// TIA Portal project "Braccio robotico_man_aut_completo_02_5AROB" (V16)

(* hardware
DEVICE "S7-1200 station_1"  S7-1200 Station
   slot 0: "Telaio di montaggio_0"  S7-1200 Rack  Rack  V1.0
   slot 1: "PLC_1"  CPU 1215C AC/DC/Rly  6ES7 215-1BG40-0XB0  V4.2
DEVICE "HMI_1"  KTP700 Basic PN
   slot 0: "HMI_1"  KTP700 Basic PN  6AV2 123-2GB03-0AX0  16.0.0.0
   slot 1: "HMI_RT_1"  KTP700 Basic PN  6AV2 123-2GB03-0AX0  16.0.0.0
   slot 5: "HMI_1.IE_CP_1"  PROFINET Interface  16.0.0.0
      slot 1: "Interfaccia_1 PROFINET"  PROFINET Interface
         slot 1: "Porta_1"  Port
*)

// ===== PLC "PLC_1"  CPU 1215C AC/DC/Rly =====

VAR_GLOBAL   // PLC tag table "Tabella variabili asse vericale"
   "SQ_alto_riferimento per lo zero" AT %I0.3 : Bool;
   "Impulsi contati dall'encoder verticale" AT %ID1000 : DWord;
   "Salita manuale" AT %M0.0 : Bool;
   "Discesa manuale" AT %M0.1 : Bool;
   "attivazione back to home" AT %M0.2 : Bool;
   "attivazione posizionamento automatico_vert" AT %M1.0 : Bool;
   "posizionamento automatico raggiunto_vert" AT %M1.1 : Bool;
   "posizionamento fuori tolleranza_vert" AT %M1.2 : Bool;
   "salita automatica" AT %M1.3 : Bool;
   "discesa automatica" AT %M1.4 : Bool;
   "Salita asse Z" AT %Q0.7 : Bool;
   "Discesa asse Z" AT %Q0.6 : Bool;
   "appoggio clock" AT %M1.6 : Bool;
   "Passo 4" AT %M30.5 : Bool;
   "Passo 5" AT %M30.6 : Bool;
   "Passo 6" AT %M30.7 : Bool;
   "Passo 7" AT %M31.0 : Bool;
   "Passo 8" AT %M31.1 : Bool;
   "Passo 9" AT %M31.2 : Bool;
   "Passo 10" AT %M31.3 : Bool;
END_VAR

VAR_GLOBAL   // PLC tag table "Tabella variabili rotazione"
   "SQ_rot_oraria_riferimento per lo zero" AT %I0.7 : Bool;
   "Impulsi contati dall'encoder rotazione" AT %ID1004 : DWord;
   "rotazione oraria manuale" AT %M2.0 : Bool;
   "rotazione antioraria manuale" AT %M2.1 : Bool;
   "attivazione back to home rotazione" AT %M2.2 : Bool;
   "attivazione posizionamento automatico_rot" AT %M3.0 : Bool;
   "posizionamento automatico raggiunto_rot" AT %M3.1 : Bool;
   "posizionamento fuori tolleranza_rot" AT %M3.2 : Bool;
   "rotazione oraria automatica" AT %M3.3 : Bool;
   "rotazione antioraria automatica" AT %M3.4 : Bool;
   "Rotazione oraria" AT %Q0.0 : Bool;
   "Rotazione antioraria" AT %Q0.1 : Bool;
END_VAR

VAR_GLOBAL   // PLC tag table "Tabella variabili braccio"
   "SQ_indietro_orizzontale" AT %I1.0 : Bool;
   "conteggio impulsi orizzontali" AT %MD5 : DInt;
   "avanti braccio manuale" AT %M4.0 : Bool;
   "indietro braccio manuale" AT %M4.1 : Bool;
   "attivazione back to home orizzontale" AT %M4.2 : Bool;
   "attivazione posizionamento automatico_orizzontale" AT %M4.3 : Bool;
   "posizionamento automatico raggiunto_orizzontale" AT %M4.4 : Bool;
   "posizionamento fuori tolleranza_orizzontale" AT %M4.5 : Bool;
   "avanti braccio in automatico" AT %M4.6 : Bool;
   "indietro braccio in automatico" AT %M4.7 : Bool;
   "Avanti braccio" AT %Q0.4 : Bool;
   "Indietro braccio" AT %Q0.5 : Bool;
   "SQ_impulsivo_orizzontale" AT %I1.1 : Bool;
END_VAR

VAR_GLOBAL   // PLC tag table "Tabella variabili pinza"
   "SQ_pinza_aperta" AT %I0.2 : Bool;
   "chiusura pinza manuale" AT %M10.0 : Bool;
   "apertura pinza manuale" AT %M10.1 : Bool;
   "attivazione back to home pinza" AT %M10.2 : Bool;
   "attivazione posizionamento automatico_pinza" AT %M10.3 : Bool;
   "posizionamento automatico raggiunto_pinza" AT %M10.4 : Bool;
   "posizionamento fuori tolleranza_pinza" AT %M10.5 : Bool;
   "chiusura pinza automatico" AT %M10.6 : Bool;
   "apertura pinza automatico" AT %M10.7 : Bool;
   "Chiusura pinza" AT %Q0.3 : Bool;
   "Apertura pinza" AT %Q0.2 : Bool;
   "conteggio impulsi pinza" AT %MD11 : DInt;
   "SQ_impulsivo_pinza" AT %I0.6 : Bool;
END_VAR

VAR_GLOBAL   // PLC tag table "Tabella variabili_ciclo_automatico"
   "condizioni_iniziali_ok" AT %M50.0 : Bool;
   "Passo 0" AT %M30.0 : Bool;
   "Passo 1" AT %M30.1 : Bool;
   "Passo 2" AT %M30.2 : Bool;
   "Passo 3" AT %M30.3 : Bool;
END_VAR

DATA_BLOCK "Blocco_dati_encoder_verticale"   // DB1
{ S7_Optimized_Access := 'TRUE' }
VERSION : 0.1
   VAR
      "posizione vericale in mm" : DInt;
      "setpoint verticale" : DInt;
      "tolleranza positiva verticale" : DInt;
      "tolleranza negativa verticale" : DInt;
      "appoggio ID1000" : DInt;
   END_VAR
BEGIN
END_DATA_BLOCK

DATA_BLOCK "Blocco_dati_HMI_verticale"   // DB2
{ S7_Optimized_Access := 'TRUE' }
VERSION : 0.1
   VAR
      jog_emergenza : Bool;
      jog_selettore_man_aut : Bool;
      jog_salita_braccio : Bool;
      jog_discesa_braccio : Bool;
      jog_back_to_home : Bool;
      setpoint_1 : DInt;
      setpoint_2 : DInt;
      setpoint_3 : DInt;
      setpoint_4 : DInt;
   END_VAR
BEGIN
END_DATA_BLOCK

DATA_BLOCK "Blocco_dati_HMI_automatico"   // DB3
{ S7_Optimized_Access := 'TRUE' }
VERSION : 0.1
   VAR
      jog_start_automatico : Bool;
      jog_ripristino : Bool;
   END_VAR
BEGIN
END_DATA_BLOCK

DATA_BLOCK "Blocco_dati_encoder_rotazione"   // DB6
{ S7_Optimized_Access := 'TRUE' }
VERSION : 0.1
   VAR
      "setpoint rotazione" : DInt;
      "tolleranza positiva rotazione" : DInt;
      "tolleranza negativa rotazione" : DInt;
      "posizione rotazione in gradi" : DInt;
      "appoggio ID1004" : DInt;
   END_VAR
BEGIN
END_DATA_BLOCK

DATA_BLOCK "Blocco_dati_HMI_rotazione"   // DB7
{ S7_Optimized_Access := 'TRUE' }
VERSION : 0.1
   VAR
      jog_rotazione_oraria : Bool;
      jog_rotazione_antioraia : Bool;
      jog_back_to_home_rotazione : Bool;
      jog_posizionamento_automatico_rot : Bool;
      setpoint_1 : DInt;
      setpoint_2 : DInt;
      setpoint_3 : DInt;
   END_VAR
BEGIN
END_DATA_BLOCK

DATA_BLOCK "Blocco_dati_contaimpulsi_braccio"   // DB8
{ S7_Optimized_Access := 'TRUE' }
VERSION : 0.1
   VAR
      "posizione orizzontale in mm" : DInt;
      "setpoint orizzontale" : DInt;
      "tolleranza positiva orizzontale" : DInt;
      "tolleranza negativa orizzontale" : DInt;
   END_VAR
BEGIN
END_DATA_BLOCK

DATA_BLOCK "Blocco_dati_contaimpulsi_pinza"   // DB9
{ S7_Optimized_Access := 'TRUE' }
VERSION : 0.1
   VAR
      "setpoint chiusura pinza" : DInt;
      "tolleranza positiva pinza" : DInt;
      "tolleranza negativa pinza" : DInt;
   END_VAR
BEGIN
END_DATA_BLOCK

DATA_BLOCK "Blocco_dati_HMI_braccio"   // DB10
{ S7_Optimized_Access := 'TRUE' }
VERSION : 0.1
   VAR
      jog_avanti_braccio : Bool;
      jog_indietro_braccio : Bool;
      jog_back_to_home_orizzontale : Bool;
      setpoint_1 : DInt;
      setpoint_2 : DInt;
      setpoint_3 : DInt;
   END_VAR
BEGIN
END_DATA_BLOCK

DATA_BLOCK "Blocco_dati_HMI_pinza"   // DB11
{ S7_Optimized_Access := 'TRUE' }
VERSION : 0.1
   VAR
      jog_chiusura_pinza : Bool;
      jog_apertura_pinza : Bool;
      jog_back_to_home_pinza : Bool;
      setpoint_1 : DInt;
      setpoint_2 : DInt;
   END_VAR
BEGIN
END_DATA_BLOCK

// folder: System blocks/Program resources

DATA_BLOCK "IEC_Counter_0_DB_1"   // DB12
{ S7_Optimized_Access := 'TRUE' }
AUTHOR : Simatic
FAMILY : IEC
NAME : CNTR
VERSION : 1.0
// stored: InstanceOfName IEC_COUNTER
"IEC_COUNTER"
BEGIN
END_DATA_BLOCK

DATA_BLOCK "TImer_passo9"   // DB13
{ S7_Optimized_Access := 'TRUE' }
AUTHOR : Simatic
FAMILY : IEC
NAME : IEC_TMR
VERSION : 1.0
// stored: InstanceOfName IEC_TIMER
"IEC_TIMER"
BEGIN
END_DATA_BLOCK

// folder: (top level)

FUNCTION "01_Calcoli_encoder_verticale" : Void   // FC1, LAD
{ S7_Optimized_Access := 'TRUE' }
VERSION : 0.1
BEGIN

REGION Network 1: Contatore veloce da configurare nelle proprietà della CPU
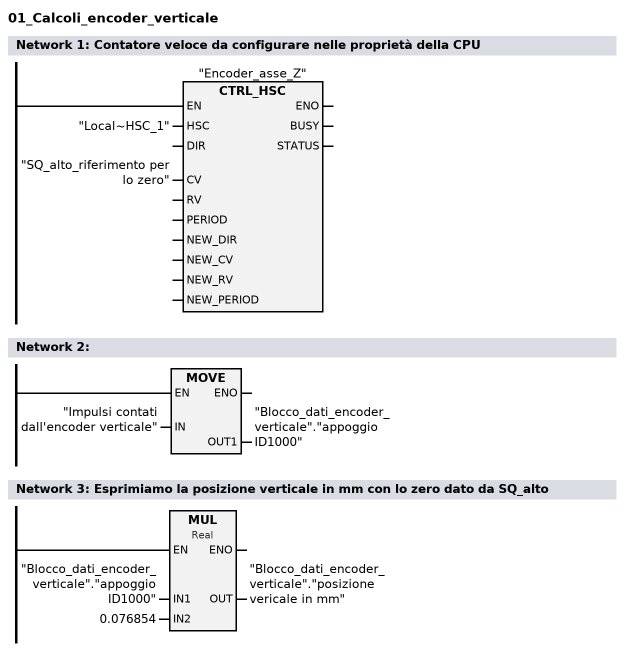
   "Encoder_asse_Z"(HSC := "Local~HSC_1", CV := "SQ_alto_riferimento per lo zero");   // CTRL_HSC
END_REGION

REGION Network 2
   RUNG wire#powerrail
      Move(in := "Impulsi contati dall'encoder verticale", out1 => "Blocco_dati_encoder_verticale"."appoggio ID1000")
   END_RUNG
   // the same network as SCL:
   "Blocco_dati_encoder_verticale"."appoggio ID1000" := "Impulsi contati dall'encoder verticale";
END_REGION

REGION Network 3: Esprimiamo la posizione verticale in mm con lo zero dato da SQ_alto
   RUNG wire#powerrail
      { S7_Templates := "SrcType := Real" } Mul(in1 := "Blocco_dati_encoder_verticale"."appoggio ID1000", in2 := 0.076854, out => "Blocco_dati_encoder_verticale"."posizione vericale in mm")
   END_RUNG
   // the same network as SCL:
   "Blocco_dati_encoder_verticale"."posizione vericale in mm" := "Blocco_dati_encoder_verticale"."appoggio ID1000" * 0.076854;
END_REGION
END_FUNCTION

FUNCTION "02_Gestione_manuale_verticale" : Void   // FC2, LAD
{ S7_Optimized_Access := 'TRUE' }
VERSION : 0.1
BEGIN

REGION Network 1: Attivazione salita in manuale
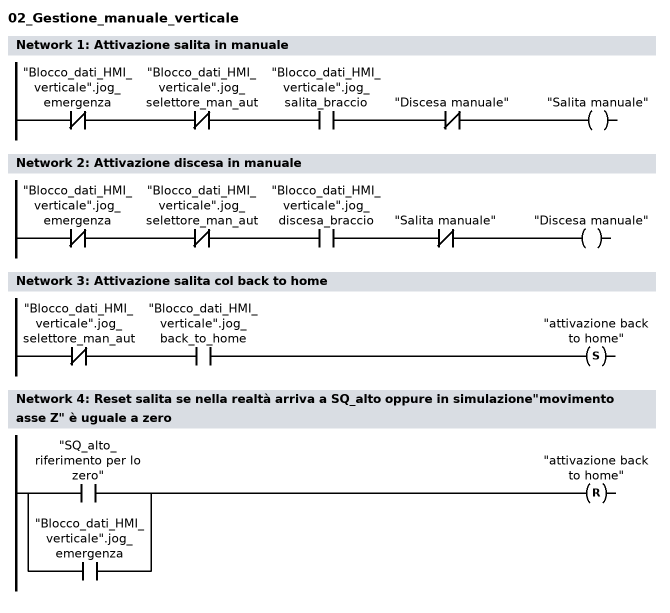
   RUNG wire#powerrail
      I_Contact( "Blocco_dati_HMI_verticale".jog_emergenza )
      I_Contact( "Blocco_dati_HMI_verticale".jog_selettore_man_aut )
      Contact( "Blocco_dati_HMI_verticale".jog_salita_braccio )
      I_Contact( "Discesa manuale" )
      Coil( "Salita manuale" )
   END_RUNG
   // the same network as SCL:
   "Salita manuale" := NOT "Blocco_dati_HMI_verticale".jog_emergenza AND NOT "Blocco_dati_HMI_verticale".jog_selettore_man_aut AND "Blocco_dati_HMI_verticale".jog_salita_braccio AND NOT "Discesa manuale";
END_REGION

REGION Network 2: Attivazione discesa in manuale
   RUNG wire#powerrail
      I_Contact( "Blocco_dati_HMI_verticale".jog_emergenza )
      I_Contact( "Blocco_dati_HMI_verticale".jog_selettore_man_aut )
      Contact( "Blocco_dati_HMI_verticale".jog_discesa_braccio )
      I_Contact( "Salita manuale" )
      Coil( "Discesa manuale" )
   END_RUNG
   // the same network as SCL:
   "Discesa manuale" := NOT "Blocco_dati_HMI_verticale".jog_emergenza AND NOT "Blocco_dati_HMI_verticale".jog_selettore_man_aut AND "Blocco_dati_HMI_verticale".jog_discesa_braccio AND NOT "Salita manuale";
END_REGION

REGION Network 3: Attivazione salita col back to home
   RUNG wire#powerrail
      I_Contact( "Blocco_dati_HMI_verticale".jog_selettore_man_aut )
      Contact( "Blocco_dati_HMI_verticale".jog_back_to_home )
      S_Coil( "attivazione back to home" )
   END_RUNG
   // the same network as SCL:
   IF NOT "Blocco_dati_HMI_verticale".jog_selettore_man_aut AND "Blocco_dati_HMI_verticale".jog_back_to_home THEN
       "attivazione back to home" := TRUE;
   END_IF;
END_REGION

REGION Network 4: Reset salita se nella realtà arriva a SQ_alto oppure in simulazione"movimento asse Z" è uguale a zero
   RUNG wire#powerrail
      Contact( "SQ_alto_riferimento per lo zero" )
      wire#w1
      R_Coil( "attivazione back to home" )
   END_RUNG
   RUNG wire#powerrail
      Contact( "Blocco_dati_HMI_verticale".jog_emergenza )
   END_RUNG wire#w1
   // the same network as SCL:
   IF "SQ_alto_riferimento per lo zero" OR "Blocco_dati_HMI_verticale".jog_emergenza THEN
       "attivazione back to home" := FALSE;
   END_IF;
END_REGION
END_FUNCTION

FUNCTION "03_Gestione_automatica_verticale" : Void   // FC3, LAD
{ S7_Optimized_Access := 'TRUE' }
VERSION : 0.1
BEGIN

REGION Network 1: Determinazione del valore della tolleranza positiva
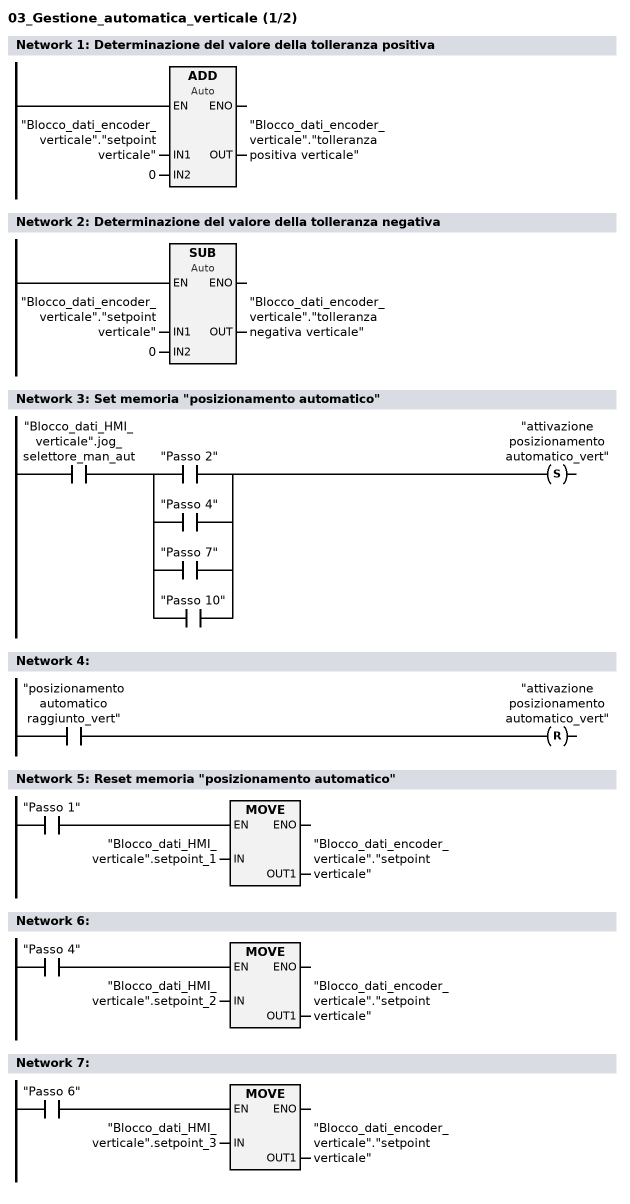
   RUNG wire#powerrail
      Add(in1 := "Blocco_dati_encoder_verticale"."setpoint verticale", in2 := 0, out => "Blocco_dati_encoder_verticale"."tolleranza positiva verticale")
   END_RUNG
   // the same network as SCL:
   "Blocco_dati_encoder_verticale"."tolleranza positiva verticale" := "Blocco_dati_encoder_verticale"."setpoint verticale" + 0;
END_REGION

REGION Network 2: Determinazione del valore della tolleranza negativa
   RUNG wire#powerrail
      Sub(in1 := "Blocco_dati_encoder_verticale"."setpoint verticale", in2 := 0, out => "Blocco_dati_encoder_verticale"."tolleranza negativa verticale")
   END_RUNG
   // the same network as SCL:
   "Blocco_dati_encoder_verticale"."tolleranza negativa verticale" := "Blocco_dati_encoder_verticale"."setpoint verticale" - 0;
END_REGION

REGION Network 3: Set memoria "posizionamento automatico"
   RUNG wire#powerrail
      Contact( "Blocco_dati_HMI_verticale".jog_selettore_man_aut )
      wire#w1
      Contact( "Passo 2" )
      wire#w2
      S_Coil( "attivazione posizionamento automatico_vert" )
   END_RUNG
   RUNG wire#w1
      Contact( "Passo 4" )
   END_RUNG wire#w2
   RUNG wire#w1
      Contact( "Passo 7" )
   END_RUNG wire#w2
   RUNG wire#w1
      Contact( "Passo 10" )
   END_RUNG wire#w2
   // the same network as SCL:
   IF "Blocco_dati_HMI_verticale".jog_selettore_man_aut AND ("Passo 2" OR "Passo 4" OR "Passo 7" OR "Passo 10") THEN
       "attivazione posizionamento automatico_vert" := TRUE;
   END_IF;
END_REGION

REGION Network 4
   RUNG wire#powerrail
      Contact( "posizionamento automatico raggiunto_vert" )
      R_Coil( "attivazione posizionamento automatico_vert" )
   END_RUNG
   // the same network as SCL:
   IF "posizionamento automatico raggiunto_vert" THEN
       "attivazione posizionamento automatico_vert" := FALSE;
   END_IF;
END_REGION

REGION Network 5: Reset memoria "posizionamento automatico"
   RUNG wire#powerrail
      Contact( "Passo 1" )
      Move(in := "Blocco_dati_HMI_verticale".setpoint_1, out1 => "Blocco_dati_encoder_verticale"."setpoint verticale")
   END_RUNG
   // the same network as SCL:
   IF "Passo 1" THEN
       "Blocco_dati_encoder_verticale"."setpoint verticale" := "Blocco_dati_HMI_verticale".setpoint_1;
   END_IF;
END_REGION

REGION Network 6
   RUNG wire#powerrail
      Contact( "Passo 4" )
      Move(in := "Blocco_dati_HMI_verticale".setpoint_2, out1 => "Blocco_dati_encoder_verticale"."setpoint verticale")
   END_RUNG
   // the same network as SCL:
   IF "Passo 4" THEN
       "Blocco_dati_encoder_verticale"."setpoint verticale" := "Blocco_dati_HMI_verticale".setpoint_2;
   END_IF;
END_REGION

REGION Network 7
   RUNG wire#powerrail
      Contact( "Passo 6" )
      Move(in := "Blocco_dati_HMI_verticale".setpoint_3, out1 => "Blocco_dati_encoder_verticale"."setpoint verticale")
   END_RUNG
   // the same network as SCL:
   IF "Passo 6" THEN
       "Blocco_dati_encoder_verticale"."setpoint verticale" := "Blocco_dati_HMI_verticale".setpoint_3;
   END_IF;
END_REGION

REGION Network 8: Posizionamento fuori tolleranza
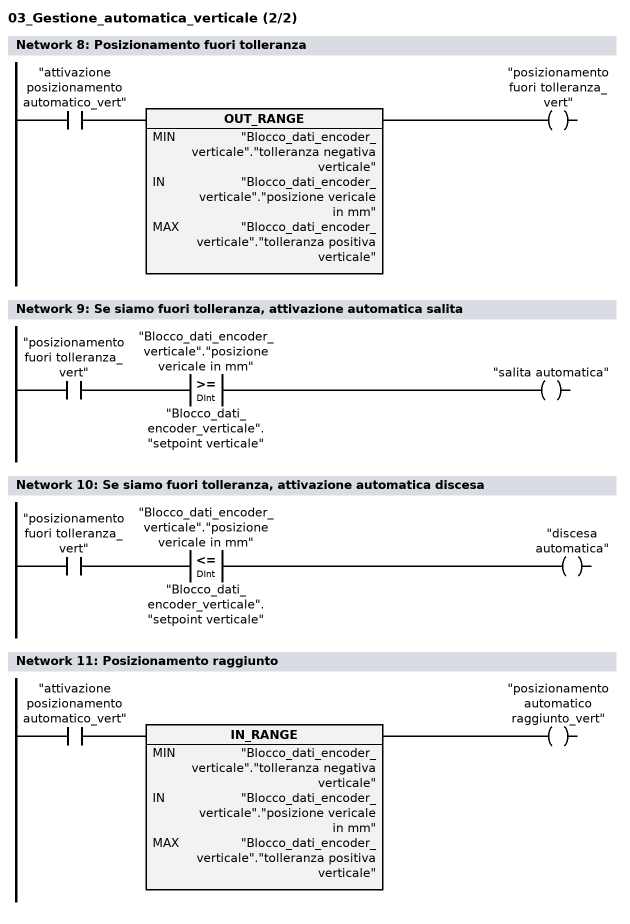
   "posizionamento fuori tolleranza_vert" := "attivazione posizionamento automatico_vert" AND (("Blocco_dati_encoder_verticale"."posizione vericale in mm" < "Blocco_dati_encoder_verticale"."tolleranza negativa verticale") OR ("Blocco_dati_encoder_verticale"."posizione vericale in mm" > "Blocco_dati_encoder_verticale"."tolleranza positiva verticale"));
END_REGION

REGION Network 9: Se siamo fuori tolleranza, attivazione automatica salita
   RUNG wire#powerrail
      Contact( "posizionamento fuori tolleranza_vert" )
      { S7_Templates := "SrcType := DInt" } GE_Contact(in1 := "Blocco_dati_encoder_verticale"."posizione vericale in mm", in2 := "Blocco_dati_encoder_verticale"."setpoint verticale")
      Coil( "salita automatica" )
   END_RUNG
   // the same network as SCL:
   "salita automatica" := "posizionamento fuori tolleranza_vert" AND ("Blocco_dati_encoder_verticale"."posizione vericale in mm" >= "Blocco_dati_encoder_verticale"."setpoint verticale");
END_REGION

REGION Network 10: Se siamo fuori tolleranza, attivazione automatica discesa
   RUNG wire#powerrail
      Contact( "posizionamento fuori tolleranza_vert" )
      { S7_Templates := "SrcType := DInt" } LE_Contact(in1 := "Blocco_dati_encoder_verticale"."posizione vericale in mm", in2 := "Blocco_dati_encoder_verticale"."setpoint verticale")
      Coil( "discesa automatica" )
   END_RUNG
   // the same network as SCL:
   "discesa automatica" := "posizionamento fuori tolleranza_vert" AND ("Blocco_dati_encoder_verticale"."posizione vericale in mm" <= "Blocco_dati_encoder_verticale"."setpoint verticale");
END_REGION

REGION Network 11: Posizionamento raggiunto
   RUNG wire#powerrail
      Contact( "attivazione posizionamento automatico_vert" )
      { S7_Templates := "SrcType := DInt" } InRange(min := "Blocco_dati_encoder_verticale"."tolleranza negativa verticale", in := "Blocco_dati_encoder_verticale"."posizione vericale in mm", max := "Blocco_dati_encoder_verticale"."tolleranza positiva verticale")
      Coil( "posizionamento automatico raggiunto_vert" )
   END_RUNG
   // the same network as SCL:
   "posizionamento automatico raggiunto_vert" := "attivazione posizionamento automatico_vert" AND ("Blocco_dati_encoder_verticale"."tolleranza negativa verticale" <= "Blocco_dati_encoder_verticale"."posizione vericale in mm") AND ("Blocco_dati_encoder_verticale"."posizione vericale in mm" <= "Blocco_dati_encoder_verticale"."tolleranza positiva verticale");
END_REGION
END_FUNCTION

FUNCTION "04_Attivazione_uscite_verticale" : Void   // FC4, LAD
{ S7_Optimized_Access := 'TRUE' }
VERSION : 0.1
BEGIN

REGION Network 1: Attivazione dell'uscita salita
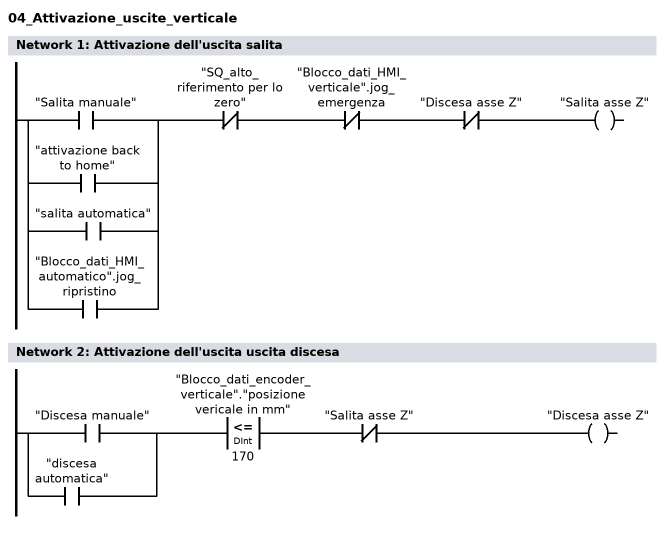
   RUNG wire#powerrail
      Contact( "Salita manuale" )
      wire#w1
      I_Contact( "SQ_alto_riferimento per lo zero" )
      I_Contact( "Blocco_dati_HMI_verticale".jog_emergenza )
      I_Contact( "Discesa asse Z" )
      Coil( "Salita asse Z" )
   END_RUNG
   RUNG wire#powerrail
      Contact( "attivazione back to home" )
   END_RUNG wire#w1
   RUNG wire#powerrail
      Contact( "salita automatica" )
   END_RUNG wire#w1
   RUNG wire#powerrail
      Contact( "Blocco_dati_HMI_automatico".jog_ripristino )
   END_RUNG wire#w1
   // the same network as SCL:
   "Salita asse Z" := ("Salita manuale" OR "attivazione back to home" OR "salita automatica" OR "Blocco_dati_HMI_automatico".jog_ripristino) AND NOT "SQ_alto_riferimento per lo zero" AND NOT "Blocco_dati_HMI_verticale".jog_emergenza AND NOT "Discesa asse Z";
END_REGION

REGION Network 2: Attivazione dell'uscita uscita discesa
   RUNG wire#powerrail
      Contact( "Discesa manuale" )
      wire#w1
      { S7_Templates := "SrcType := DInt" } LE_Contact(in1 := "Blocco_dati_encoder_verticale"."posizione vericale in mm", in2 := 170)
      I_Contact( "Salita asse Z" )
      Coil( "Discesa asse Z" )
   END_RUNG
   RUNG wire#powerrail
      Contact( "discesa automatica" )
   END_RUNG wire#w1
   // the same network as SCL:
   "Discesa asse Z" := ("Discesa manuale" OR "discesa automatica") AND ("Blocco_dati_encoder_verticale"."posizione vericale in mm" <= 170) AND NOT "Salita asse Z";
END_REGION
END_FUNCTION

FUNCTION "05_Calcoli_encoder_rotazione" : Void   // FC5, LAD
{ S7_Optimized_Access := 'TRUE' }
VERSION : 0.1
BEGIN

REGION Network 1: Contatore veloce da configurare nelle proprietà della CPU
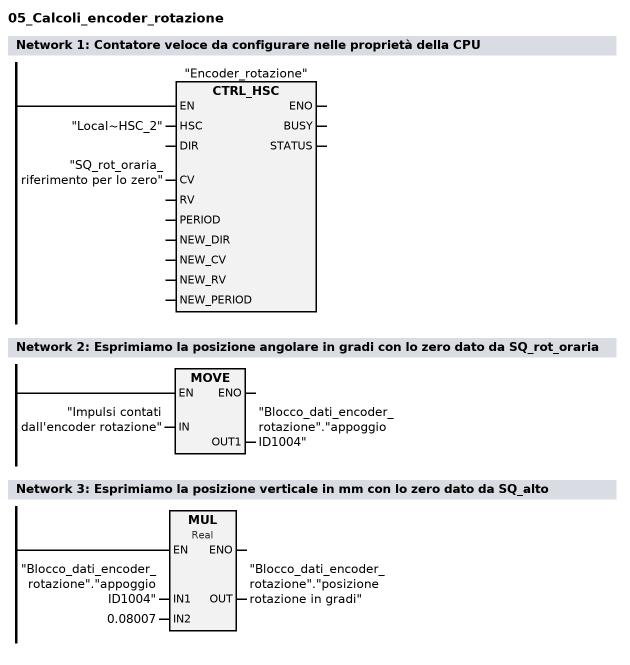
   "Encoder_rotazione"(HSC := "Local~HSC_2", CV := "SQ_rot_oraria_riferimento per lo zero");   // CTRL_HSC
END_REGION

REGION Network 2: Esprimiamo la posizione angolare in gradi con lo zero dato da SQ_rot_oraria
   RUNG wire#powerrail
      Move(in := "Impulsi contati dall'encoder rotazione", out1 => "Blocco_dati_encoder_rotazione"."appoggio ID1004")
   END_RUNG
   // the same network as SCL:
   "Blocco_dati_encoder_rotazione"."appoggio ID1004" := "Impulsi contati dall'encoder rotazione";
END_REGION

REGION Network 3: Esprimiamo la posizione verticale in mm con lo zero dato da SQ_alto
   RUNG wire#powerrail
      { S7_Templates := "SrcType := Real" } Mul(in1 := "Blocco_dati_encoder_rotazione"."appoggio ID1004", in2 := 0.08007, out => "Blocco_dati_encoder_rotazione"."posizione rotazione in gradi")
   END_RUNG
   // the same network as SCL:
   "Blocco_dati_encoder_rotazione"."posizione rotazione in gradi" := "Blocco_dati_encoder_rotazione"."appoggio ID1004" * 0.08007;
END_REGION
END_FUNCTION

FUNCTION "06_Gestione_manuale_rotazione" : Void   // FC6, LAD
{ S7_Optimized_Access := 'TRUE' }
VERSION : 0.1
BEGIN

REGION Network 1: Attivazione salita in manuale
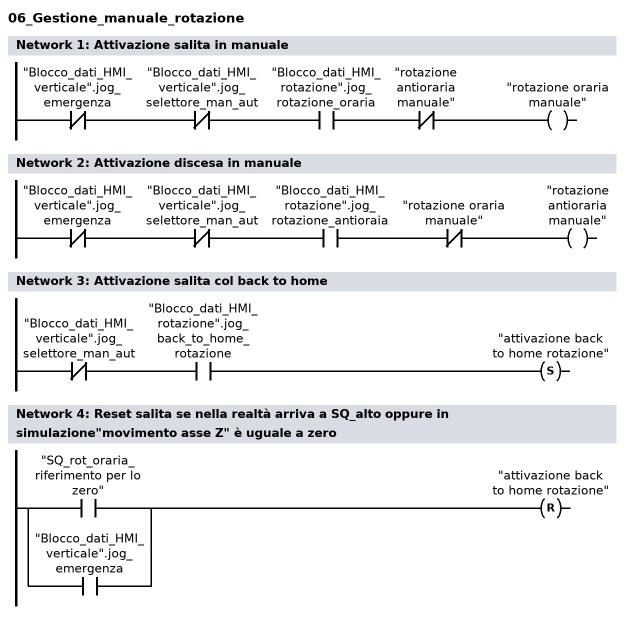
   RUNG wire#powerrail
      I_Contact( "Blocco_dati_HMI_verticale".jog_emergenza )
      I_Contact( "Blocco_dati_HMI_verticale".jog_selettore_man_aut )
      Contact( "Blocco_dati_HMI_rotazione".jog_rotazione_oraria )
      I_Contact( "rotazione antioraria manuale" )
      Coil( "rotazione oraria manuale" )
   END_RUNG
   // the same network as SCL:
   "rotazione oraria manuale" := NOT "Blocco_dati_HMI_verticale".jog_emergenza AND NOT "Blocco_dati_HMI_verticale".jog_selettore_man_aut AND "Blocco_dati_HMI_rotazione".jog_rotazione_oraria AND NOT "rotazione antioraria manuale";
END_REGION

REGION Network 2: Attivazione discesa in manuale
   RUNG wire#powerrail
      I_Contact( "Blocco_dati_HMI_verticale".jog_emergenza )
      I_Contact( "Blocco_dati_HMI_verticale".jog_selettore_man_aut )
      Contact( "Blocco_dati_HMI_rotazione".jog_rotazione_antioraia )
      I_Contact( "rotazione oraria manuale" )
      Coil( "rotazione antioraria manuale" )
   END_RUNG
   // the same network as SCL:
   "rotazione antioraria manuale" := NOT "Blocco_dati_HMI_verticale".jog_emergenza AND NOT "Blocco_dati_HMI_verticale".jog_selettore_man_aut AND "Blocco_dati_HMI_rotazione".jog_rotazione_antioraia AND NOT "rotazione oraria manuale";
END_REGION

REGION Network 3: Attivazione salita col back to home
   RUNG wire#powerrail
      I_Contact( "Blocco_dati_HMI_verticale".jog_selettore_man_aut )
      Contact( "Blocco_dati_HMI_rotazione".jog_back_to_home_rotazione )
      S_Coil( "attivazione back to home rotazione" )
   END_RUNG
   // the same network as SCL:
   IF NOT "Blocco_dati_HMI_verticale".jog_selettore_man_aut AND "Blocco_dati_HMI_rotazione".jog_back_to_home_rotazione THEN
       "attivazione back to home rotazione" := TRUE;
   END_IF;
END_REGION

REGION Network 4: Reset salita se nella realtà arriva a SQ_alto oppure in simulazione"movimento asse Z" è uguale a zero
   RUNG wire#powerrail
      Contact( "SQ_rot_oraria_riferimento per lo zero" )
      wire#w1
      R_Coil( "attivazione back to home rotazione" )
   END_RUNG
   RUNG wire#powerrail
      Contact( "Blocco_dati_HMI_verticale".jog_emergenza )
   END_RUNG wire#w1
   // the same network as SCL:
   IF "SQ_rot_oraria_riferimento per lo zero" OR "Blocco_dati_HMI_verticale".jog_emergenza THEN
       "attivazione back to home rotazione" := FALSE;
   END_IF;
END_REGION
END_FUNCTION

FUNCTION "07_Gestione_automatica_rotazione" : Void   // FC7, LAD
{ S7_Optimized_Access := 'TRUE' }
VERSION : 0.1
BEGIN

REGION Network 1: Determinazione del valore della tolleranza positiva
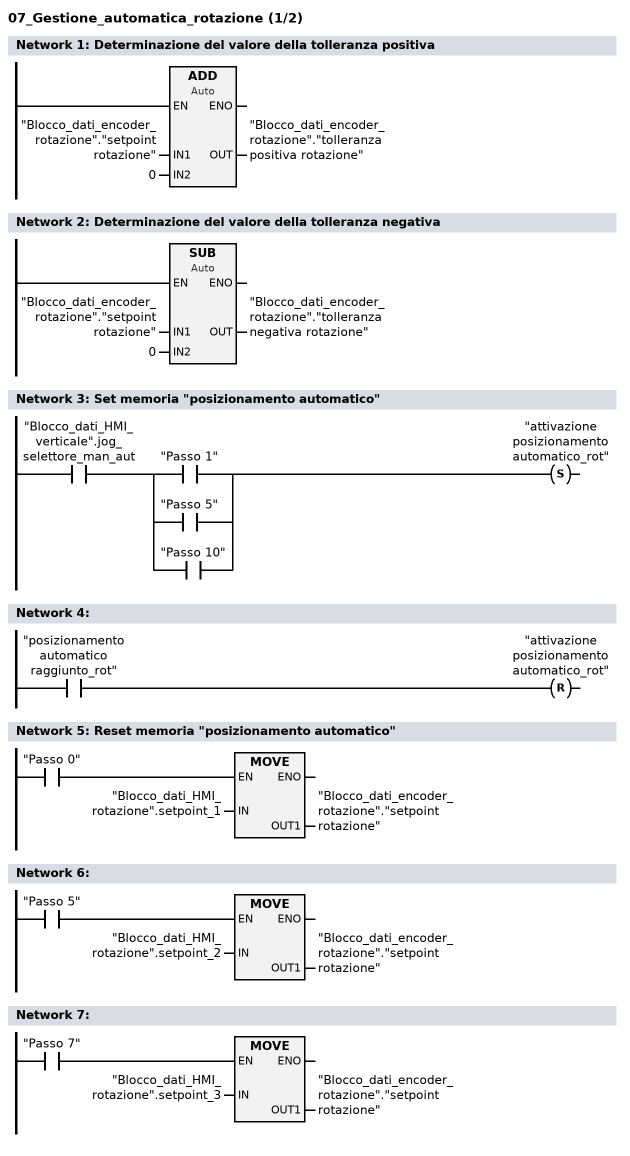
   RUNG wire#powerrail
      Add(in1 := "Blocco_dati_encoder_rotazione"."setpoint rotazione", in2 := 0, out => "Blocco_dati_encoder_rotazione"."tolleranza positiva rotazione")
   END_RUNG
   // the same network as SCL:
   "Blocco_dati_encoder_rotazione"."tolleranza positiva rotazione" := "Blocco_dati_encoder_rotazione"."setpoint rotazione" + 0;
END_REGION

REGION Network 2: Determinazione del valore della tolleranza negativa
   RUNG wire#powerrail
      Sub(in1 := "Blocco_dati_encoder_rotazione"."setpoint rotazione", in2 := 0, out => "Blocco_dati_encoder_rotazione"."tolleranza negativa rotazione")
   END_RUNG
   // the same network as SCL:
   "Blocco_dati_encoder_rotazione"."tolleranza negativa rotazione" := "Blocco_dati_encoder_rotazione"."setpoint rotazione" - 0;
END_REGION

REGION Network 3: Set memoria "posizionamento automatico"
   RUNG wire#powerrail
      Contact( "Blocco_dati_HMI_verticale".jog_selettore_man_aut )
      wire#w1
      Contact( "Passo 1" )
      wire#w2
      S_Coil( "attivazione posizionamento automatico_rot" )
   END_RUNG
   RUNG wire#w1
      Contact( "Passo 5" )
   END_RUNG wire#w2
   RUNG wire#w1
      Contact( "Passo 10" )
   END_RUNG wire#w2
   // the same network as SCL:
   IF "Blocco_dati_HMI_verticale".jog_selettore_man_aut AND ("Passo 1" OR "Passo 5" OR "Passo 10") THEN
       "attivazione posizionamento automatico_rot" := TRUE;
   END_IF;
END_REGION

REGION Network 4
   RUNG wire#powerrail
      Contact( "posizionamento automatico raggiunto_rot" )
      R_Coil( "attivazione posizionamento automatico_rot" )
   END_RUNG
   // the same network as SCL:
   IF "posizionamento automatico raggiunto_rot" THEN
       "attivazione posizionamento automatico_rot" := FALSE;
   END_IF;
END_REGION

REGION Network 5: Reset memoria "posizionamento automatico"
   RUNG wire#powerrail
      Contact( "Passo 0" )
      Move(in := "Blocco_dati_HMI_rotazione".setpoint_1, out1 => "Blocco_dati_encoder_rotazione"."setpoint rotazione")
   END_RUNG
   // the same network as SCL:
   IF "Passo 0" THEN
       "Blocco_dati_encoder_rotazione"."setpoint rotazione" := "Blocco_dati_HMI_rotazione".setpoint_1;
   END_IF;
END_REGION

REGION Network 6
   RUNG wire#powerrail
      Contact( "Passo 5" )
      Move(in := "Blocco_dati_HMI_rotazione".setpoint_2, out1 => "Blocco_dati_encoder_rotazione"."setpoint rotazione")
   END_RUNG
   // the same network as SCL:
   IF "Passo 5" THEN
       "Blocco_dati_encoder_rotazione"."setpoint rotazione" := "Blocco_dati_HMI_rotazione".setpoint_2;
   END_IF;
END_REGION

REGION Network 7
   RUNG wire#powerrail
      Contact( "Passo 7" )
      Move(in := "Blocco_dati_HMI_rotazione".setpoint_3, out1 => "Blocco_dati_encoder_rotazione"."setpoint rotazione")
   END_RUNG
   // the same network as SCL:
   IF "Passo 7" THEN
       "Blocco_dati_encoder_rotazione"."setpoint rotazione" := "Blocco_dati_HMI_rotazione".setpoint_3;
   END_IF;
END_REGION

REGION Network 8: Posizionamento fuori tolleranza
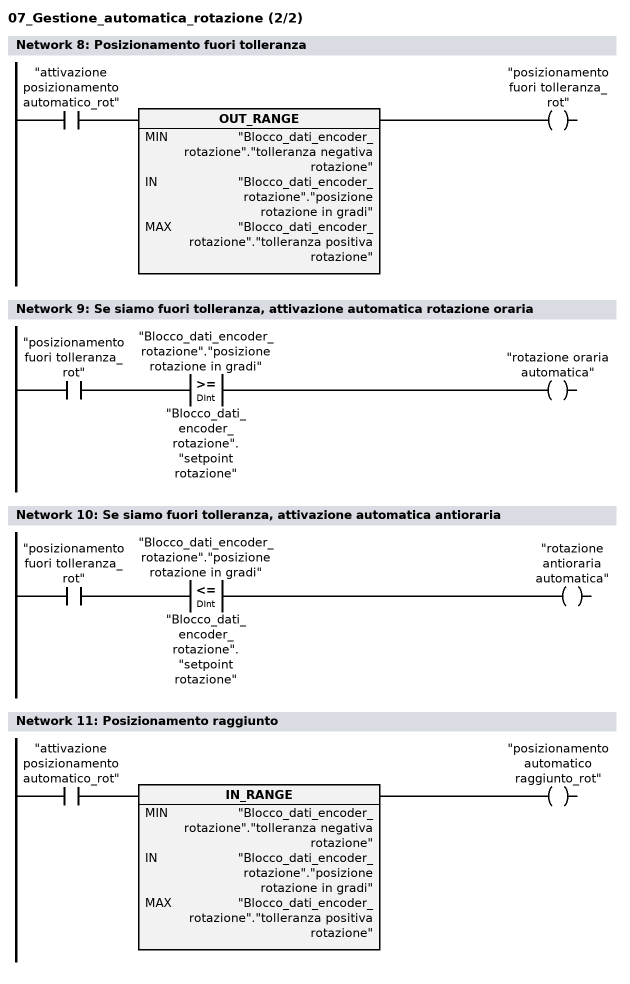
   "posizionamento fuori tolleranza_rot" := "attivazione posizionamento automatico_rot" AND (("Blocco_dati_encoder_rotazione"."posizione rotazione in gradi" < "Blocco_dati_encoder_rotazione"."tolleranza negativa rotazione") OR ("Blocco_dati_encoder_rotazione"."posizione rotazione in gradi" > "Blocco_dati_encoder_rotazione"."tolleranza positiva rotazione"));
END_REGION

REGION Network 9: Se siamo fuori tolleranza, attivazione automatica rotazione oraria
   RUNG wire#powerrail
      Contact( "posizionamento fuori tolleranza_rot" )
      { S7_Templates := "SrcType := DInt" } GE_Contact(in1 := "Blocco_dati_encoder_rotazione"."posizione rotazione in gradi", in2 := "Blocco_dati_encoder_rotazione"."setpoint rotazione")
      Coil( "rotazione oraria automatica" )
   END_RUNG
   // the same network as SCL:
   "rotazione oraria automatica" := "posizionamento fuori tolleranza_rot" AND ("Blocco_dati_encoder_rotazione"."posizione rotazione in gradi" >= "Blocco_dati_encoder_rotazione"."setpoint rotazione");
END_REGION

REGION Network 10: Se siamo fuori tolleranza, attivazione automatica antioraria
   RUNG wire#powerrail
      Contact( "posizionamento fuori tolleranza_rot" )
      { S7_Templates := "SrcType := DInt" } LE_Contact(in1 := "Blocco_dati_encoder_rotazione"."posizione rotazione in gradi", in2 := "Blocco_dati_encoder_rotazione"."setpoint rotazione")
      Coil( "rotazione antioraria automatica" )
   END_RUNG
   // the same network as SCL:
   "rotazione antioraria automatica" := "posizionamento fuori tolleranza_rot" AND ("Blocco_dati_encoder_rotazione"."posizione rotazione in gradi" <= "Blocco_dati_encoder_rotazione"."setpoint rotazione");
END_REGION

REGION Network 11: Posizionamento raggiunto
   RUNG wire#powerrail
      Contact( "attivazione posizionamento automatico_rot" )
      { S7_Templates := "SrcType := DInt" } InRange(min := "Blocco_dati_encoder_rotazione"."tolleranza negativa rotazione", in := "Blocco_dati_encoder_rotazione"."posizione rotazione in gradi", max := "Blocco_dati_encoder_rotazione"."tolleranza positiva rotazione")
      Coil( "posizionamento automatico raggiunto_rot" )
   END_RUNG
   // the same network as SCL:
   "posizionamento automatico raggiunto_rot" := "attivazione posizionamento automatico_rot" AND ("Blocco_dati_encoder_rotazione"."tolleranza negativa rotazione" <= "Blocco_dati_encoder_rotazione"."posizione rotazione in gradi") AND ("Blocco_dati_encoder_rotazione"."posizione rotazione in gradi" <= "Blocco_dati_encoder_rotazione"."tolleranza positiva rotazione");
END_REGION
END_FUNCTION

FUNCTION "08_Attivazione_uscite_rotazione" : Void   // FC8, LAD
{ S7_Optimized_Access := 'TRUE' }
VERSION : 0.1
BEGIN

REGION Network 1: Attivazione dell'uscita salita
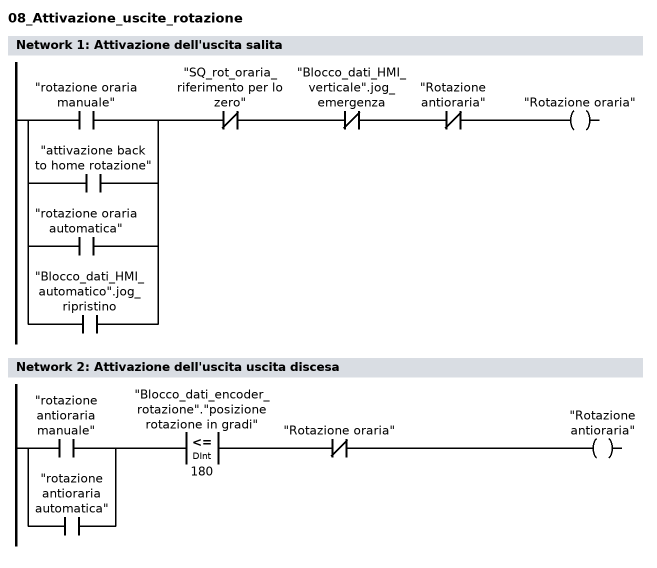
   RUNG wire#powerrail
      Contact( "rotazione oraria manuale" )
      wire#w1
      I_Contact( "SQ_rot_oraria_riferimento per lo zero" )
      I_Contact( "Blocco_dati_HMI_verticale".jog_emergenza )
      I_Contact( "Rotazione antioraria" )
      Coil( "Rotazione oraria" )
   END_RUNG
   RUNG wire#powerrail
      Contact( "attivazione back to home rotazione" )
   END_RUNG wire#w1
   RUNG wire#powerrail
      Contact( "rotazione oraria automatica" )
   END_RUNG wire#w1
   RUNG wire#powerrail
      Contact( "Blocco_dati_HMI_automatico".jog_ripristino )
   END_RUNG wire#w1
   // the same network as SCL:
   "Rotazione oraria" := ("rotazione oraria manuale" OR "attivazione back to home rotazione" OR "rotazione oraria automatica" OR "Blocco_dati_HMI_automatico".jog_ripristino) AND NOT "SQ_rot_oraria_riferimento per lo zero" AND NOT "Blocco_dati_HMI_verticale".jog_emergenza AND NOT "Rotazione antioraria";
END_REGION

REGION Network 2: Attivazione dell'uscita uscita discesa
   RUNG wire#powerrail
      Contact( "rotazione antioraria manuale" )
      wire#w1
      { S7_Templates := "SrcType := DInt" } LE_Contact(in1 := "Blocco_dati_encoder_rotazione"."posizione rotazione in gradi", in2 := 180)
      I_Contact( "Rotazione oraria" )
      Coil( "Rotazione antioraria" )
   END_RUNG
   RUNG wire#powerrail
      Contact( "rotazione antioraria automatica" )
   END_RUNG wire#w1
   // the same network as SCL:
   "Rotazione antioraria" := ("rotazione antioraria manuale" OR "rotazione antioraria automatica") AND ("Blocco_dati_encoder_rotazione"."posizione rotazione in gradi" <= 180) AND NOT "Rotazione oraria";
END_REGION
END_FUNCTION

FUNCTION "09_Calcoli_posizione_braccio" : Void   // FC9, LAD
{ S7_Optimized_Access := 'TRUE' }
VERSION : 0.1
BEGIN

REGION Network 1: Incremento conteggio degli impulsi prodotti dalla rotazione della ruota dentata caletta sulla vite senza fine del riduttore di velocità del motore braccio
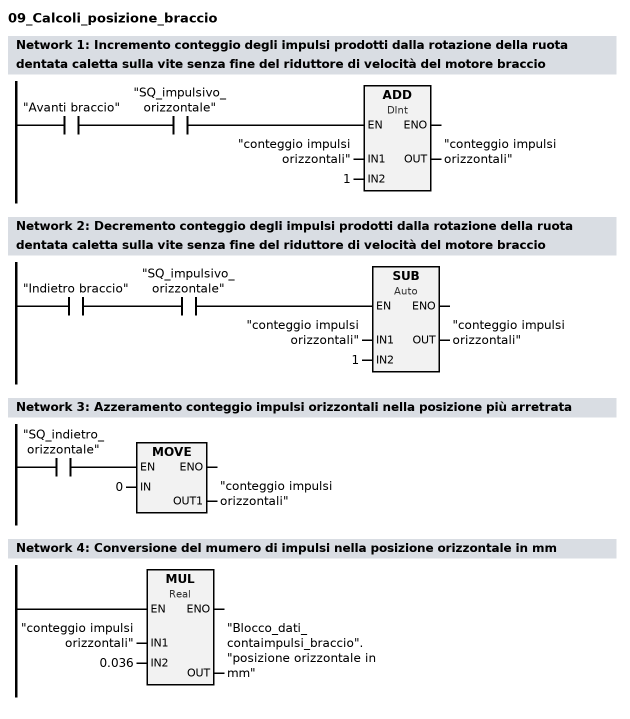
   RUNG wire#powerrail
      Contact( "Avanti braccio" )
      Contact( "SQ_impulsivo_orizzontale" )
      { S7_Templates := "SrcType := DInt" } Add(in1 := "conteggio impulsi orizzontali", in2 := 1, out => "conteggio impulsi orizzontali")
   END_RUNG
   // the same network as SCL:
   IF "Avanti braccio" AND "SQ_impulsivo_orizzontale" THEN
       "conteggio impulsi orizzontali" := "conteggio impulsi orizzontali" + 1;
   END_IF;
END_REGION

REGION Network 2: Decremento conteggio degli impulsi prodotti dalla rotazione della ruota dentata caletta sulla vite senza fine del riduttore di velocità del motore braccio
   RUNG wire#powerrail
      Contact( "Indietro braccio" )
      Contact( "SQ_impulsivo_orizzontale" )
      Sub(in1 := "conteggio impulsi orizzontali", in2 := 1, out => "conteggio impulsi orizzontali")
   END_RUNG
   // the same network as SCL:
   IF "Indietro braccio" AND "SQ_impulsivo_orizzontale" THEN
       "conteggio impulsi orizzontali" := "conteggio impulsi orizzontali" - 1;
   END_IF;
END_REGION

REGION Network 3: Azzeramento conteggio impulsi orizzontali nella posizione più arretrata
   RUNG wire#powerrail
      Contact( "SQ_indietro_orizzontale" )
      Move(in := 0, out1 => "conteggio impulsi orizzontali")
   END_RUNG
   // the same network as SCL:
   IF "SQ_indietro_orizzontale" THEN "conteggio impulsi orizzontali" := 0; END_IF;
END_REGION

REGION Network 4: Conversione del mumero di impulsi nella posizione orizzontale in mm
   RUNG wire#powerrail
      { S7_Templates := "SrcType := Real" } Mul(in1 := "conteggio impulsi orizzontali", in2 := 0.036, out => "Blocco_dati_contaimpulsi_braccio"."posizione orizzontale in mm")
   END_RUNG
   // the same network as SCL:
   "Blocco_dati_contaimpulsi_braccio"."posizione orizzontale in mm" := "conteggio impulsi orizzontali" * 0.036;
END_REGION
END_FUNCTION

FUNCTION "13_Calcoli_posizione_pinza" : Void   // FC10, LAD
{ S7_Optimized_Access := 'TRUE' }
VERSION : 0.1
BEGIN

REGION Network 1
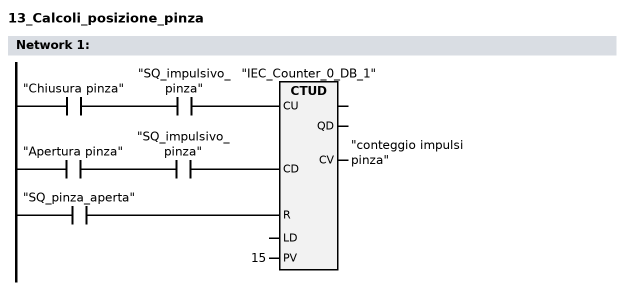
   "IEC_Counter_0_DB_1".CTUD(CU := "Chiusura pinza" AND "SQ_impulsivo_pinza",
                           CD := "Apertura pinza" AND "SQ_impulsivo_pinza",
                           R := "SQ_pinza_aperta",
                           PV := 15,
                           CV => "conteggio impulsi pinza");
END_REGION
END_FUNCTION

FUNCTION "10_Gestione_manuale_braccio" : Void   // FC11, LAD
{ S7_Optimized_Access := 'TRUE' }
VERSION : 0.1
BEGIN

REGION Network 1: Attivazione indietro braccio in manuale
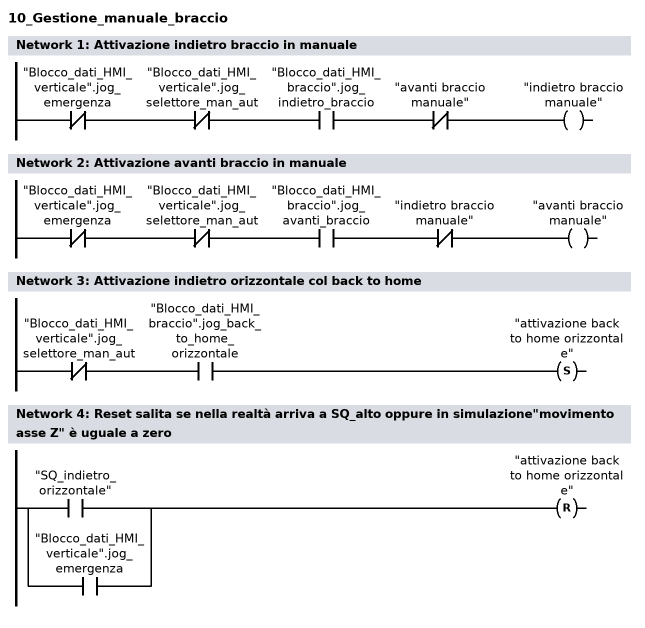
   RUNG wire#powerrail
      I_Contact( "Blocco_dati_HMI_verticale".jog_emergenza )
      I_Contact( "Blocco_dati_HMI_verticale".jog_selettore_man_aut )
      Contact( "Blocco_dati_HMI_braccio".jog_indietro_braccio )
      I_Contact( "avanti braccio manuale" )
      Coil( "indietro braccio manuale" )
   END_RUNG
   // the same network as SCL:
   "indietro braccio manuale" := NOT "Blocco_dati_HMI_verticale".jog_emergenza AND NOT "Blocco_dati_HMI_verticale".jog_selettore_man_aut AND "Blocco_dati_HMI_braccio".jog_indietro_braccio AND NOT "avanti braccio manuale";
END_REGION

REGION Network 2: Attivazione avanti braccio in manuale
   RUNG wire#powerrail
      I_Contact( "Blocco_dati_HMI_verticale".jog_emergenza )
      I_Contact( "Blocco_dati_HMI_verticale".jog_selettore_man_aut )
      Contact( "Blocco_dati_HMI_braccio".jog_avanti_braccio )
      I_Contact( "indietro braccio manuale" )
      Coil( "avanti braccio manuale" )
   END_RUNG
   // the same network as SCL:
   "avanti braccio manuale" := NOT "Blocco_dati_HMI_verticale".jog_emergenza AND NOT "Blocco_dati_HMI_verticale".jog_selettore_man_aut AND "Blocco_dati_HMI_braccio".jog_avanti_braccio AND NOT "indietro braccio manuale";
END_REGION

REGION Network 3: Attivazione indietro orizzontale col back to home
   RUNG wire#powerrail
      I_Contact( "Blocco_dati_HMI_verticale".jog_selettore_man_aut )
      Contact( "Blocco_dati_HMI_braccio".jog_back_to_home_orizzontale )
      S_Coil( "attivazione back to home orizzontale" )
   END_RUNG
   // the same network as SCL:
   IF NOT "Blocco_dati_HMI_verticale".jog_selettore_man_aut AND "Blocco_dati_HMI_braccio".jog_back_to_home_orizzontale THEN
       "attivazione back to home orizzontale" := TRUE;
   END_IF;
END_REGION

REGION Network 4: Reset salita se nella realtà arriva a SQ_alto oppure in simulazione"movimento asse Z" è uguale a zero
   RUNG wire#powerrail
      Contact( "SQ_indietro_orizzontale" )
      wire#w1
      R_Coil( "attivazione back to home orizzontale" )
   END_RUNG
   RUNG wire#powerrail
      Contact( "Blocco_dati_HMI_verticale".jog_emergenza )
   END_RUNG wire#w1
   // the same network as SCL:
   IF "SQ_indietro_orizzontale" OR "Blocco_dati_HMI_verticale".jog_emergenza THEN
       "attivazione back to home orizzontale" := FALSE;
   END_IF;
END_REGION
END_FUNCTION

FUNCTION "14_Gestione_manuale_pinza" : Void   // FC12, LAD
{ S7_Optimized_Access := 'TRUE' }
VERSION : 0.1
BEGIN

REGION Network 1: Attivazione indietro braccio in manuale
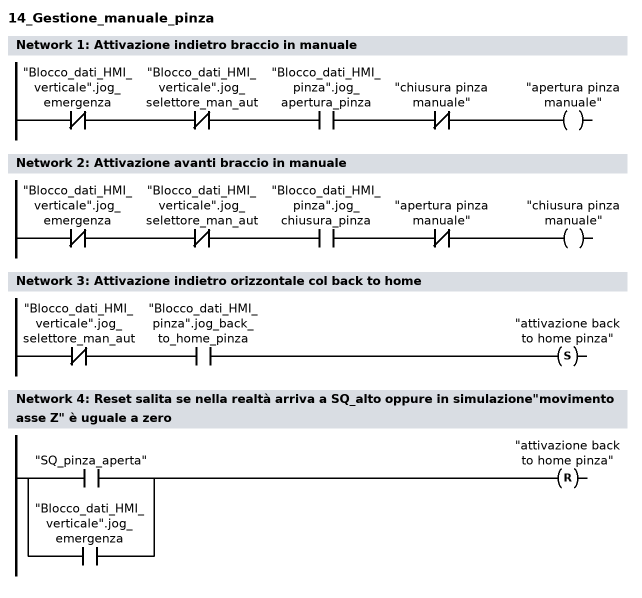
   RUNG wire#powerrail
      I_Contact( "Blocco_dati_HMI_verticale".jog_emergenza )
      I_Contact( "Blocco_dati_HMI_verticale".jog_selettore_man_aut )
      Contact( "Blocco_dati_HMI_pinza".jog_apertura_pinza )
      I_Contact( "chiusura pinza manuale" )
      Coil( "apertura pinza manuale" )
   END_RUNG
   // the same network as SCL:
   "apertura pinza manuale" := NOT "Blocco_dati_HMI_verticale".jog_emergenza AND NOT "Blocco_dati_HMI_verticale".jog_selettore_man_aut AND "Blocco_dati_HMI_pinza".jog_apertura_pinza AND NOT "chiusura pinza manuale";
END_REGION

REGION Network 2: Attivazione avanti braccio in manuale
   RUNG wire#powerrail
      I_Contact( "Blocco_dati_HMI_verticale".jog_emergenza )
      I_Contact( "Blocco_dati_HMI_verticale".jog_selettore_man_aut )
      Contact( "Blocco_dati_HMI_pinza".jog_chiusura_pinza )
      I_Contact( "apertura pinza manuale" )
      Coil( "chiusura pinza manuale" )
   END_RUNG
   // the same network as SCL:
   "chiusura pinza manuale" := NOT "Blocco_dati_HMI_verticale".jog_emergenza AND NOT "Blocco_dati_HMI_verticale".jog_selettore_man_aut AND "Blocco_dati_HMI_pinza".jog_chiusura_pinza AND NOT "apertura pinza manuale";
END_REGION

REGION Network 3: Attivazione indietro orizzontale col back to home
   RUNG wire#powerrail
      I_Contact( "Blocco_dati_HMI_verticale".jog_selettore_man_aut )
      Contact( "Blocco_dati_HMI_pinza".jog_back_to_home_pinza )
      S_Coil( "attivazione back to home pinza" )
   END_RUNG
   // the same network as SCL:
   IF NOT "Blocco_dati_HMI_verticale".jog_selettore_man_aut AND "Blocco_dati_HMI_pinza".jog_back_to_home_pinza THEN
       "attivazione back to home pinza" := TRUE;
   END_IF;
END_REGION

REGION Network 4: Reset salita se nella realtà arriva a SQ_alto oppure in simulazione"movimento asse Z" è uguale a zero
   RUNG wire#powerrail
      Contact( "SQ_pinza_aperta" )
      wire#w1
      R_Coil( "attivazione back to home pinza" )
   END_RUNG
   RUNG wire#powerrail
      Contact( "Blocco_dati_HMI_verticale".jog_emergenza )
   END_RUNG wire#w1
   // the same network as SCL:
   IF "SQ_pinza_aperta" OR "Blocco_dati_HMI_verticale".jog_emergenza THEN
       "attivazione back to home pinza" := FALSE;
   END_IF;
END_REGION
END_FUNCTION

FUNCTION "11_Gestione_automatica_braccio" : Void   // FC13, LAD
{ S7_Optimized_Access := 'TRUE' }
VERSION : 0.1
BEGIN

REGION Network 1: Determinazione del valore della tolleranza positiva
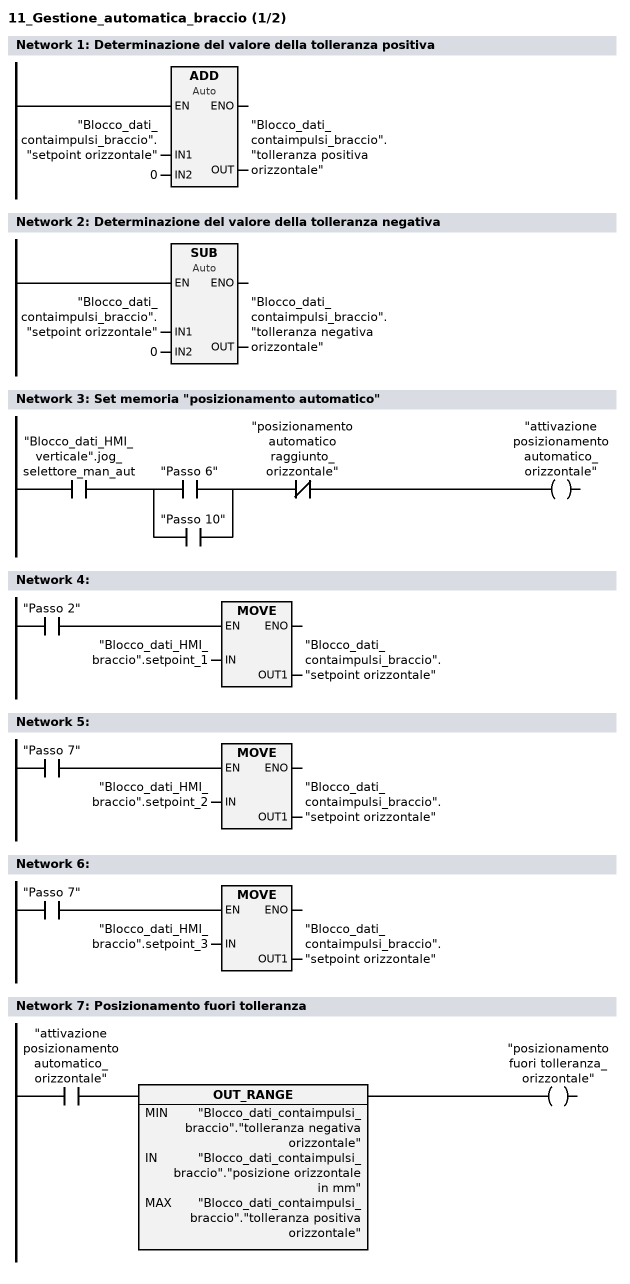
   RUNG wire#powerrail
      Add(in1 := "Blocco_dati_contaimpulsi_braccio"."setpoint orizzontale", in2 := 0, out => "Blocco_dati_contaimpulsi_braccio"."tolleranza positiva orizzontale")
   END_RUNG
   // the same network as SCL:
   "Blocco_dati_contaimpulsi_braccio"."tolleranza positiva orizzontale" := "Blocco_dati_contaimpulsi_braccio"."setpoint orizzontale" + 0;
END_REGION

REGION Network 2: Determinazione del valore della tolleranza negativa
   RUNG wire#powerrail
      Sub(in1 := "Blocco_dati_contaimpulsi_braccio"."setpoint orizzontale", in2 := 0, out => "Blocco_dati_contaimpulsi_braccio"."tolleranza negativa orizzontale")
   END_RUNG
   // the same network as SCL:
   "Blocco_dati_contaimpulsi_braccio"."tolleranza negativa orizzontale" := "Blocco_dati_contaimpulsi_braccio"."setpoint orizzontale" - 0;
END_REGION

REGION Network 3: Set memoria "posizionamento automatico"
   RUNG wire#powerrail
      Contact( "Blocco_dati_HMI_verticale".jog_selettore_man_aut )
      wire#w1
      Contact( "Passo 6" )
      wire#w2
      I_Contact( "posizionamento automatico raggiunto_orizzontale" )
      Coil( "attivazione posizionamento automatico_orizzontale" )
   END_RUNG
   RUNG wire#w1
      Contact( "Passo 10" )
   END_RUNG wire#w2
   // the same network as SCL:
   "attivazione posizionamento automatico_orizzontale" := "Blocco_dati_HMI_verticale".jog_selettore_man_aut AND ("Passo 6" OR "Passo 10") AND NOT "posizionamento automatico raggiunto_orizzontale";
END_REGION

REGION Network 4
   RUNG wire#powerrail
      Contact( "Passo 2" )
      Move(in := "Blocco_dati_HMI_braccio".setpoint_1, out1 => "Blocco_dati_contaimpulsi_braccio"."setpoint orizzontale")
   END_RUNG
   // the same network as SCL:
   IF "Passo 2" THEN
       "Blocco_dati_contaimpulsi_braccio"."setpoint orizzontale" := "Blocco_dati_HMI_braccio".setpoint_1;
   END_IF;
END_REGION

REGION Network 5
   RUNG wire#powerrail
      Contact( "Passo 7" )
      Move(in := "Blocco_dati_HMI_braccio".setpoint_2, out1 => "Blocco_dati_contaimpulsi_braccio"."setpoint orizzontale")
   END_RUNG
   // the same network as SCL:
   IF "Passo 7" THEN
       "Blocco_dati_contaimpulsi_braccio"."setpoint orizzontale" := "Blocco_dati_HMI_braccio".setpoint_2;
   END_IF;
END_REGION

REGION Network 6
   RUNG wire#powerrail
      Contact( "Passo 7" )
      Move(in := "Blocco_dati_HMI_braccio".setpoint_3, out1 => "Blocco_dati_contaimpulsi_braccio"."setpoint orizzontale")
   END_RUNG
   // the same network as SCL:
   IF "Passo 7" THEN
       "Blocco_dati_contaimpulsi_braccio"."setpoint orizzontale" := "Blocco_dati_HMI_braccio".setpoint_3;
   END_IF;
END_REGION

REGION Network 7: Posizionamento fuori tolleranza
   "posizionamento fuori tolleranza_orizzontale" := "attivazione posizionamento automatico_orizzontale" AND (("Blocco_dati_contaimpulsi_braccio"."posizione orizzontale in mm" < "Blocco_dati_contaimpulsi_braccio"."tolleranza negativa orizzontale") OR ("Blocco_dati_contaimpulsi_braccio"."posizione orizzontale in mm" > "Blocco_dati_contaimpulsi_braccio"."tolleranza positiva orizzontale"));
END_REGION

REGION Network 8: Se siamo fuori tolleranza, attivazione automatica indietro braccio
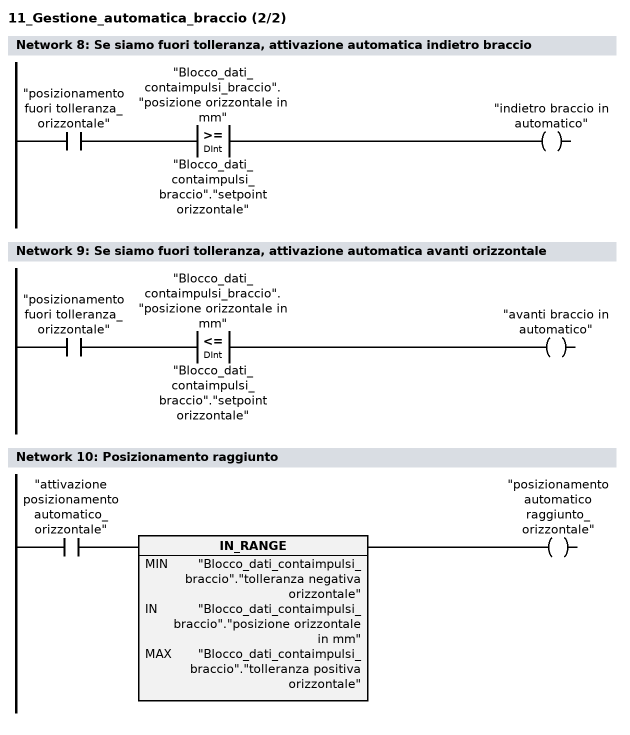
   RUNG wire#powerrail
      Contact( "posizionamento fuori tolleranza_orizzontale" )
      { S7_Templates := "SrcType := DInt" } GE_Contact(in1 := "Blocco_dati_contaimpulsi_braccio"."posizione orizzontale in mm", in2 := "Blocco_dati_contaimpulsi_braccio"."setpoint orizzontale")
      Coil( "indietro braccio in automatico" )
   END_RUNG
   // the same network as SCL:
   "indietro braccio in automatico" := "posizionamento fuori tolleranza_orizzontale" AND ("Blocco_dati_contaimpulsi_braccio"."posizione orizzontale in mm" >= "Blocco_dati_contaimpulsi_braccio"."setpoint orizzontale");
END_REGION

REGION Network 9: Se siamo fuori tolleranza, attivazione automatica avanti orizzontale
   RUNG wire#powerrail
      Contact( "posizionamento fuori tolleranza_orizzontale" )
      { S7_Templates := "SrcType := DInt" } LE_Contact(in1 := "Blocco_dati_contaimpulsi_braccio"."posizione orizzontale in mm", in2 := "Blocco_dati_contaimpulsi_braccio"."setpoint orizzontale")
      Coil( "avanti braccio in automatico" )
   END_RUNG
   // the same network as SCL:
   "avanti braccio in automatico" := "posizionamento fuori tolleranza_orizzontale" AND ("Blocco_dati_contaimpulsi_braccio"."posizione orizzontale in mm" <= "Blocco_dati_contaimpulsi_braccio"."setpoint orizzontale");
END_REGION

REGION Network 10: Posizionamento raggiunto
   RUNG wire#powerrail
      Contact( "attivazione posizionamento automatico_orizzontale" )
      { S7_Templates := "SrcType := DInt" } InRange(min := "Blocco_dati_contaimpulsi_braccio"."tolleranza negativa orizzontale", in := "Blocco_dati_contaimpulsi_braccio"."posizione orizzontale in mm", max := "Blocco_dati_contaimpulsi_braccio"."tolleranza positiva orizzontale")
      Coil( "posizionamento automatico raggiunto_orizzontale" )
   END_RUNG
   // the same network as SCL:
   "posizionamento automatico raggiunto_orizzontale" := "attivazione posizionamento automatico_orizzontale" AND ("Blocco_dati_contaimpulsi_braccio"."tolleranza negativa orizzontale" <= "Blocco_dati_contaimpulsi_braccio"."posizione orizzontale in mm") AND ("Blocco_dati_contaimpulsi_braccio"."posizione orizzontale in mm" <= "Blocco_dati_contaimpulsi_braccio"."tolleranza positiva orizzontale");
END_REGION
END_FUNCTION

FUNCTION "15_Gestione_automatica_pinza" : Void   // FC14, LAD
{ S7_Optimized_Access := 'TRUE' }
VERSION : 0.1
BEGIN

REGION Network 1: Determinazione del valore della tolleranza positiva
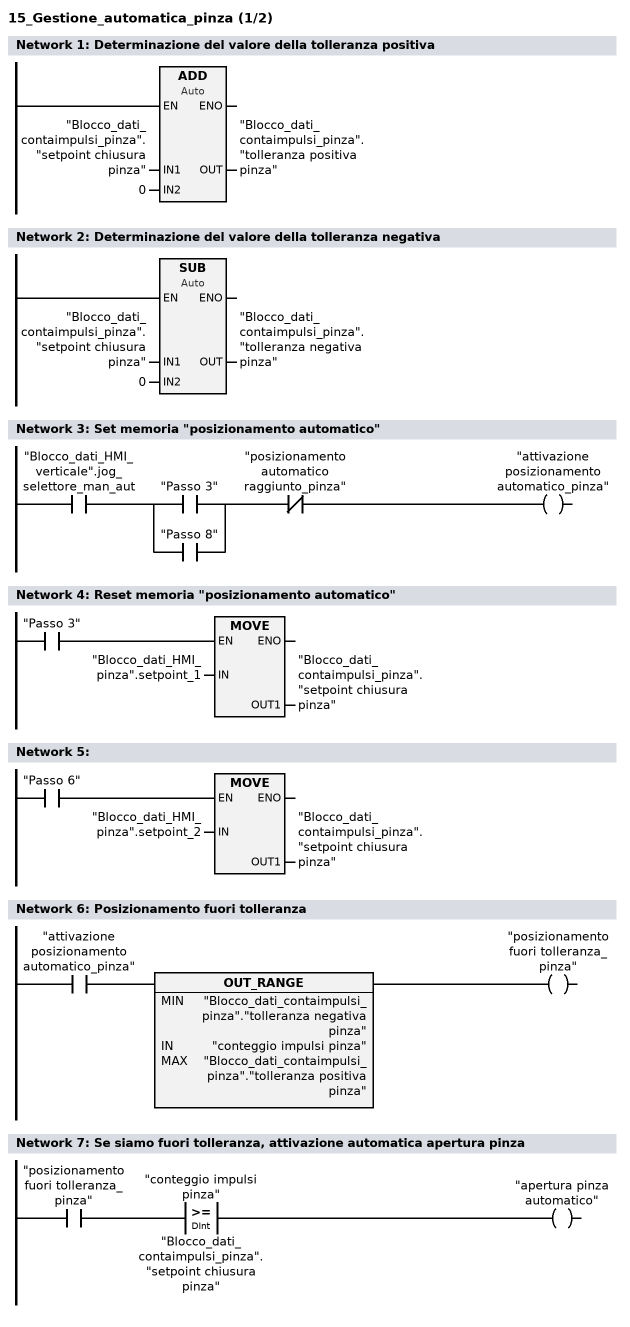
   RUNG wire#powerrail
      Add(in1 := "Blocco_dati_contaimpulsi_pinza"."setpoint chiusura pinza", in2 := 0, out => "Blocco_dati_contaimpulsi_pinza"."tolleranza positiva pinza")
   END_RUNG
   // the same network as SCL:
   "Blocco_dati_contaimpulsi_pinza"."tolleranza positiva pinza" := "Blocco_dati_contaimpulsi_pinza"."setpoint chiusura pinza" + 0;
END_REGION

REGION Network 2: Determinazione del valore della tolleranza negativa
   RUNG wire#powerrail
      Sub(in1 := "Blocco_dati_contaimpulsi_pinza"."setpoint chiusura pinza", in2 := 0, out => "Blocco_dati_contaimpulsi_pinza"."tolleranza negativa pinza")
   END_RUNG
   // the same network as SCL:
   "Blocco_dati_contaimpulsi_pinza"."tolleranza negativa pinza" := "Blocco_dati_contaimpulsi_pinza"."setpoint chiusura pinza" - 0;
END_REGION

REGION Network 3: Set memoria "posizionamento automatico"
   RUNG wire#powerrail
      Contact( "Blocco_dati_HMI_verticale".jog_selettore_man_aut )
      wire#w1
      Contact( "Passo 3" )
      wire#w2
      I_Contact( "posizionamento automatico raggiunto_pinza" )
      Coil( "attivazione posizionamento automatico_pinza" )
   END_RUNG
   RUNG wire#w1
      Contact( "Passo 8" )
   END_RUNG wire#w2
   // the same network as SCL:
   "attivazione posizionamento automatico_pinza" := "Blocco_dati_HMI_verticale".jog_selettore_man_aut AND ("Passo 3" OR "Passo 8") AND NOT "posizionamento automatico raggiunto_pinza";
END_REGION

REGION Network 4: Reset memoria "posizionamento automatico"
   RUNG wire#powerrail
      Contact( "Passo 3" )
      Move(in := "Blocco_dati_HMI_pinza".setpoint_1, out1 => "Blocco_dati_contaimpulsi_pinza"."setpoint chiusura pinza")
   END_RUNG
   // the same network as SCL:
   IF "Passo 3" THEN
       "Blocco_dati_contaimpulsi_pinza"."setpoint chiusura pinza" := "Blocco_dati_HMI_pinza".setpoint_1;
   END_IF;
END_REGION

REGION Network 5
   RUNG wire#powerrail
      Contact( "Passo 6" )
      Move(in := "Blocco_dati_HMI_pinza".setpoint_2, out1 => "Blocco_dati_contaimpulsi_pinza"."setpoint chiusura pinza")
   END_RUNG
   // the same network as SCL:
   IF "Passo 6" THEN
       "Blocco_dati_contaimpulsi_pinza"."setpoint chiusura pinza" := "Blocco_dati_HMI_pinza".setpoint_2;
   END_IF;
END_REGION

REGION Network 6: Posizionamento fuori tolleranza
   "posizionamento fuori tolleranza_pinza" := "attivazione posizionamento automatico_pinza" AND (("conteggio impulsi pinza" < "Blocco_dati_contaimpulsi_pinza"."tolleranza negativa pinza") OR ("conteggio impulsi pinza" > "Blocco_dati_contaimpulsi_pinza"."tolleranza positiva pinza"));
END_REGION

REGION Network 7: Se siamo fuori tolleranza, attivazione automatica apertura pinza
   RUNG wire#powerrail
      Contact( "posizionamento fuori tolleranza_pinza" )
      { S7_Templates := "SrcType := DInt" } GE_Contact(in1 := "conteggio impulsi pinza", in2 := "Blocco_dati_contaimpulsi_pinza"."setpoint chiusura pinza")
      Coil( "apertura pinza automatico" )
   END_RUNG
   // the same network as SCL:
   "apertura pinza automatico" := "posizionamento fuori tolleranza_pinza" AND ("conteggio impulsi pinza" >= "Blocco_dati_contaimpulsi_pinza"."setpoint chiusura pinza");
END_REGION

REGION Network 8: Se siamo fuori tolleranza, attivazione automatica chiusura pinza
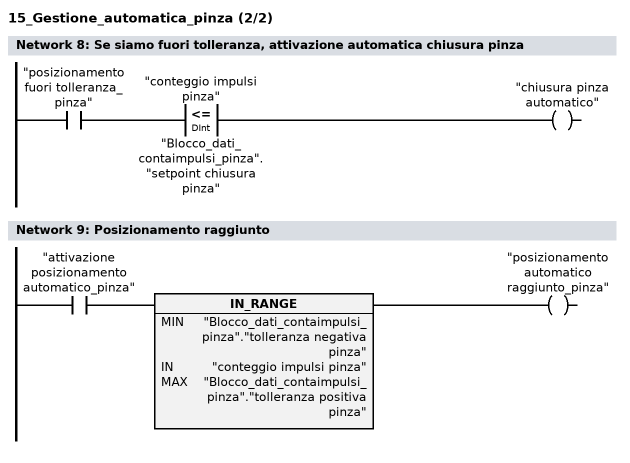
   RUNG wire#powerrail
      Contact( "posizionamento fuori tolleranza_pinza" )
      { S7_Templates := "SrcType := DInt" } LE_Contact(in1 := "conteggio impulsi pinza", in2 := "Blocco_dati_contaimpulsi_pinza"."setpoint chiusura pinza")
      Coil( "chiusura pinza automatico" )
   END_RUNG
   // the same network as SCL:
   "chiusura pinza automatico" := "posizionamento fuori tolleranza_pinza" AND ("conteggio impulsi pinza" <= "Blocco_dati_contaimpulsi_pinza"."setpoint chiusura pinza");
END_REGION

REGION Network 9: Posizionamento raggiunto
   RUNG wire#powerrail
      Contact( "attivazione posizionamento automatico_pinza" )
      { S7_Templates := "SrcType := DInt" } InRange(min := "Blocco_dati_contaimpulsi_pinza"."tolleranza negativa pinza", in := "conteggio impulsi pinza", max := "Blocco_dati_contaimpulsi_pinza"."tolleranza positiva pinza")
      Coil( "posizionamento automatico raggiunto_pinza" )
   END_RUNG
   // the same network as SCL:
   "posizionamento automatico raggiunto_pinza" := "attivazione posizionamento automatico_pinza" AND ("Blocco_dati_contaimpulsi_pinza"."tolleranza negativa pinza" <= "conteggio impulsi pinza") AND ("conteggio impulsi pinza" <= "Blocco_dati_contaimpulsi_pinza"."tolleranza positiva pinza");
END_REGION
END_FUNCTION

FUNCTION "16_Attivazione_uscite_pinza" : Void   // FC15, LAD
{ S7_Optimized_Access := 'TRUE' }
VERSION : 0.1
BEGIN

REGION Network 1: Attivazione dell'uscita salita
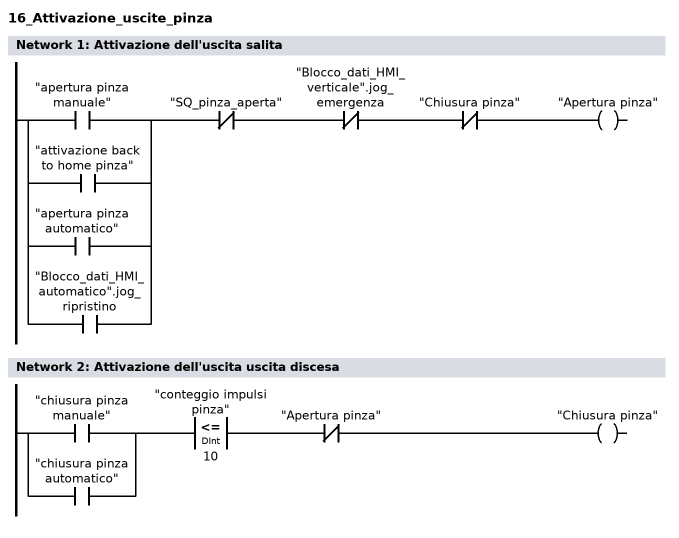
   RUNG wire#powerrail
      Contact( "apertura pinza manuale" )
      wire#w1
      I_Contact( "SQ_pinza_aperta" )
      I_Contact( "Blocco_dati_HMI_verticale".jog_emergenza )
      I_Contact( "Chiusura pinza" )
      Coil( "Apertura pinza" )
   END_RUNG
   RUNG wire#powerrail
      Contact( "attivazione back to home pinza" )
   END_RUNG wire#w1
   RUNG wire#powerrail
      Contact( "apertura pinza automatico" )
   END_RUNG wire#w1
   RUNG wire#powerrail
      Contact( "Blocco_dati_HMI_automatico".jog_ripristino )
   END_RUNG wire#w1
   // the same network as SCL:
   "Apertura pinza" := ("apertura pinza manuale" OR "attivazione back to home pinza" OR "apertura pinza automatico" OR "Blocco_dati_HMI_automatico".jog_ripristino) AND NOT "SQ_pinza_aperta" AND NOT "Blocco_dati_HMI_verticale".jog_emergenza AND NOT "Chiusura pinza";
END_REGION

REGION Network 2: Attivazione dell'uscita uscita discesa
   RUNG wire#powerrail
      Contact( "chiusura pinza manuale" )
      wire#w1
      { S7_Templates := "SrcType := DInt" } LE_Contact(in1 := "conteggio impulsi pinza", in2 := 10)
      I_Contact( "Apertura pinza" )
      Coil( "Chiusura pinza" )
   END_RUNG
   RUNG wire#powerrail
      Contact( "chiusura pinza automatico" )
   END_RUNG wire#w1
   // the same network as SCL:
   "Chiusura pinza" := ("chiusura pinza manuale" OR "chiusura pinza automatico") AND ("conteggio impulsi pinza" <= 10) AND NOT "Apertura pinza";
END_REGION
END_FUNCTION

FUNCTION "12_Attivazione_uscite_braccio" : Void   // FC16, LAD
{ S7_Optimized_Access := 'TRUE' }
VERSION : 0.1
BEGIN

REGION Network 1: Attivazione dell'uscita salita
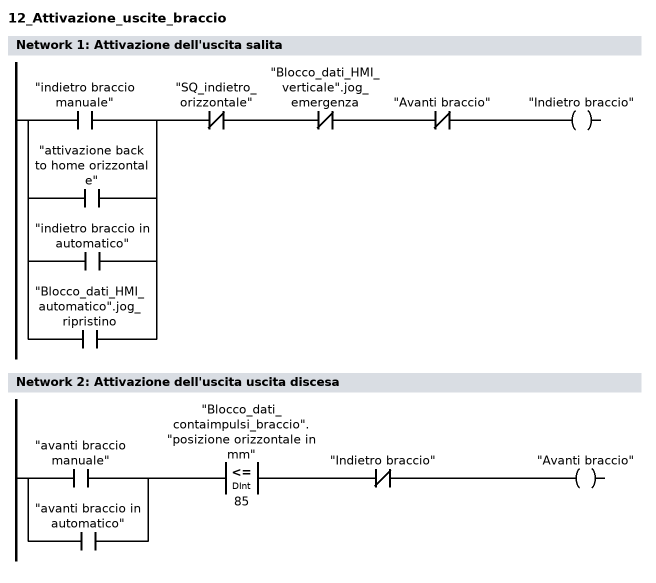
   RUNG wire#powerrail
      Contact( "indietro braccio manuale" )
      wire#w1
      I_Contact( "SQ_indietro_orizzontale" )
      I_Contact( "Blocco_dati_HMI_verticale".jog_emergenza )
      I_Contact( "Avanti braccio" )
      Coil( "Indietro braccio" )
   END_RUNG
   RUNG wire#powerrail
      Contact( "attivazione back to home orizzontale" )
   END_RUNG wire#w1
   RUNG wire#powerrail
      Contact( "indietro braccio in automatico" )
   END_RUNG wire#w1
   RUNG wire#powerrail
      Contact( "Blocco_dati_HMI_automatico".jog_ripristino )
   END_RUNG wire#w1
   // the same network as SCL:
   "Indietro braccio" := ("indietro braccio manuale" OR "attivazione back to home orizzontale" OR "indietro braccio in automatico" OR "Blocco_dati_HMI_automatico".jog_ripristino) AND NOT "SQ_indietro_orizzontale" AND NOT "Blocco_dati_HMI_verticale".jog_emergenza AND NOT "Avanti braccio";
END_REGION

REGION Network 2: Attivazione dell'uscita uscita discesa
   RUNG wire#powerrail
      Contact( "avanti braccio manuale" )
      wire#w1
      { S7_Templates := "SrcType := DInt" } LE_Contact(in1 := "Blocco_dati_contaimpulsi_braccio"."posizione orizzontale in mm", in2 := 85)
      I_Contact( "Indietro braccio" )
      Coil( "Avanti braccio" )
   END_RUNG
   RUNG wire#powerrail
      Contact( "avanti braccio in automatico" )
   END_RUNG wire#w1
   // the same network as SCL:
   "Avanti braccio" := ("avanti braccio manuale" OR "avanti braccio in automatico") AND ("Blocco_dati_contaimpulsi_braccio"."posizione orizzontale in mm" <= 85) AND NOT "Indietro braccio";
END_REGION
END_FUNCTION

FUNCTION "Ciclo_automatico_1" : Void   // FC17, LAD
{ S7_Optimized_Access := 'TRUE' }
VERSION : 0.1
BEGIN

REGION Network 1
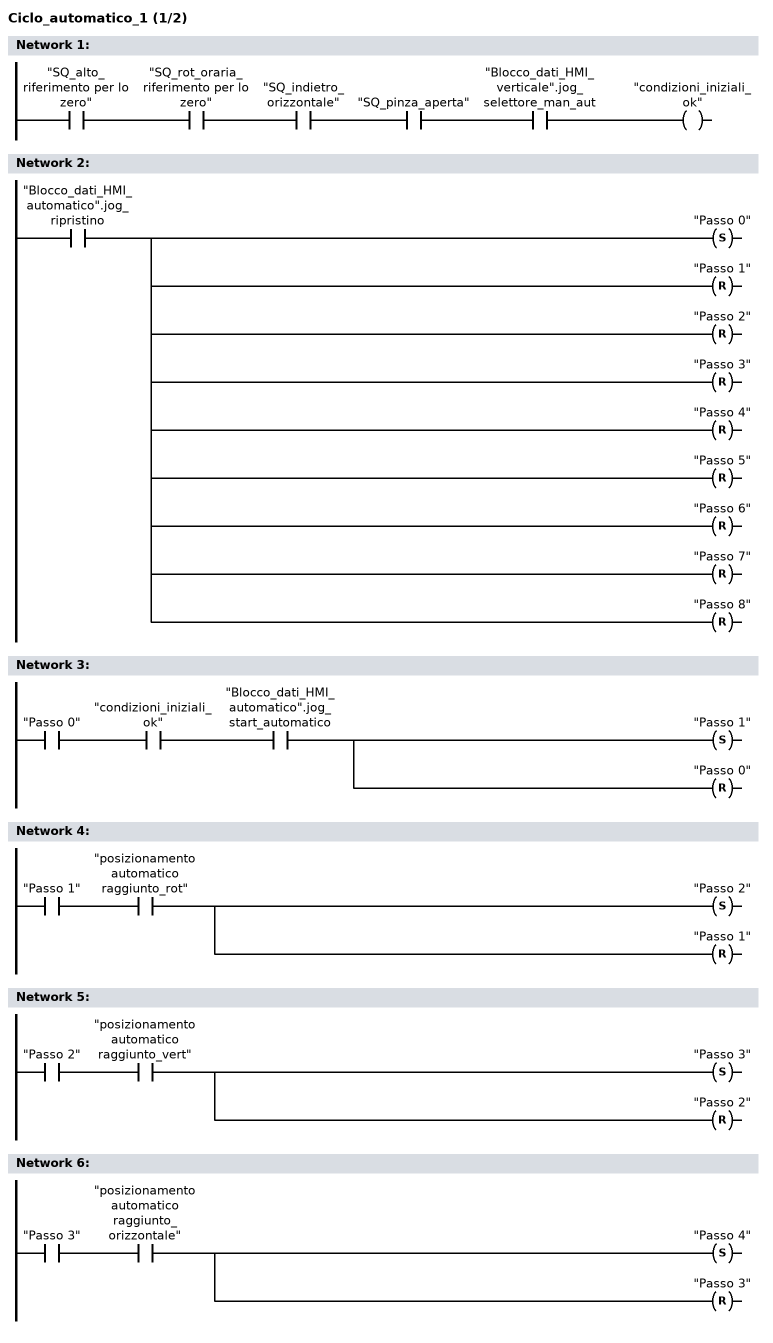
   RUNG wire#powerrail
      Contact( "SQ_alto_riferimento per lo zero" )
      Contact( "SQ_rot_oraria_riferimento per lo zero" )
      Contact( "SQ_indietro_orizzontale" )
      Contact( "SQ_pinza_aperta" )
      Contact( "Blocco_dati_HMI_verticale".jog_selettore_man_aut )
      Coil( "condizioni_iniziali_ok" )
   END_RUNG
   // the same network as SCL:
   "condizioni_iniziali_ok" := "SQ_alto_riferimento per lo zero" AND "SQ_rot_oraria_riferimento per lo zero" AND "SQ_indietro_orizzontale" AND "SQ_pinza_aperta" AND "Blocco_dati_HMI_verticale".jog_selettore_man_aut;
END_REGION

REGION Network 2
   RUNG wire#powerrail
      Contact( "Blocco_dati_HMI_automatico".jog_ripristino )
      wire#w1
      S_Coil( "Passo 0" )
   END_RUNG
   RUNG wire#w1
      R_Coil( "Passo 1" )
   END_RUNG
   RUNG wire#w1
      R_Coil( "Passo 2" )
   END_RUNG
   RUNG wire#w1
      R_Coil( "Passo 3" )
   END_RUNG
   RUNG wire#w1
      R_Coil( "Passo 4" )
   END_RUNG
   RUNG wire#w1
      R_Coil( "Passo 5" )
   END_RUNG
   RUNG wire#w1
      R_Coil( "Passo 6" )
   END_RUNG
   RUNG wire#w1
      R_Coil( "Passo 7" )
   END_RUNG
   RUNG wire#w1
      R_Coil( "Passo 8" )
   END_RUNG
   // the same network as SCL:
   IF "Blocco_dati_HMI_automatico".jog_ripristino THEN
       "Passo 0" := TRUE;
       "Passo 1" := FALSE;
       "Passo 2" := FALSE;
       "Passo 3" := FALSE;
       "Passo 4" := FALSE;
       "Passo 5" := FALSE;
       "Passo 6" := FALSE;
       "Passo 7" := FALSE;
       "Passo 8" := FALSE;
   END_IF;
END_REGION

REGION Network 3
   RUNG wire#powerrail
      Contact( "Passo 0" )
      Contact( "condizioni_iniziali_ok" )
      Contact( "Blocco_dati_HMI_automatico".jog_start_automatico )
      wire#w1
      S_Coil( "Passo 1" )
   END_RUNG
   RUNG wire#w1
      R_Coil( "Passo 0" )
   END_RUNG
   // the same network as SCL:
   IF "Passo 0" AND "condizioni_iniziali_ok" AND "Blocco_dati_HMI_automatico".jog_start_automatico THEN
       "Passo 1" := TRUE;
       "Passo 0" := FALSE;
   END_IF;
END_REGION

REGION Network 4
   RUNG wire#powerrail
      Contact( "Passo 1" )
      Contact( "posizionamento automatico raggiunto_rot" )
      wire#w1
      S_Coil( "Passo 2" )
   END_RUNG
   RUNG wire#w1
      R_Coil( "Passo 1" )
   END_RUNG
   // the same network as SCL:
   IF "Passo 1" AND "posizionamento automatico raggiunto_rot" THEN
       "Passo 2" := TRUE;
       "Passo 1" := FALSE;
   END_IF;
END_REGION

REGION Network 5
   RUNG wire#powerrail
      Contact( "Passo 2" )
      Contact( "posizionamento automatico raggiunto_vert" )
      wire#w1
      S_Coil( "Passo 3" )
   END_RUNG
   RUNG wire#w1
      R_Coil( "Passo 2" )
   END_RUNG
   // the same network as SCL:
   IF "Passo 2" AND "posizionamento automatico raggiunto_vert" THEN
       "Passo 3" := TRUE;
       "Passo 2" := FALSE;
   END_IF;
END_REGION

REGION Network 6
   RUNG wire#powerrail
      Contact( "Passo 3" )
      Contact( "posizionamento automatico raggiunto_orizzontale" )
      wire#w1
      S_Coil( "Passo 4" )
   END_RUNG
   RUNG wire#w1
      R_Coil( "Passo 3" )
   END_RUNG
   // the same network as SCL:
   IF "Passo 3" AND "posizionamento automatico raggiunto_orizzontale" THEN
       "Passo 4" := TRUE;
       "Passo 3" := FALSE;
   END_IF;
END_REGION

REGION Network 7
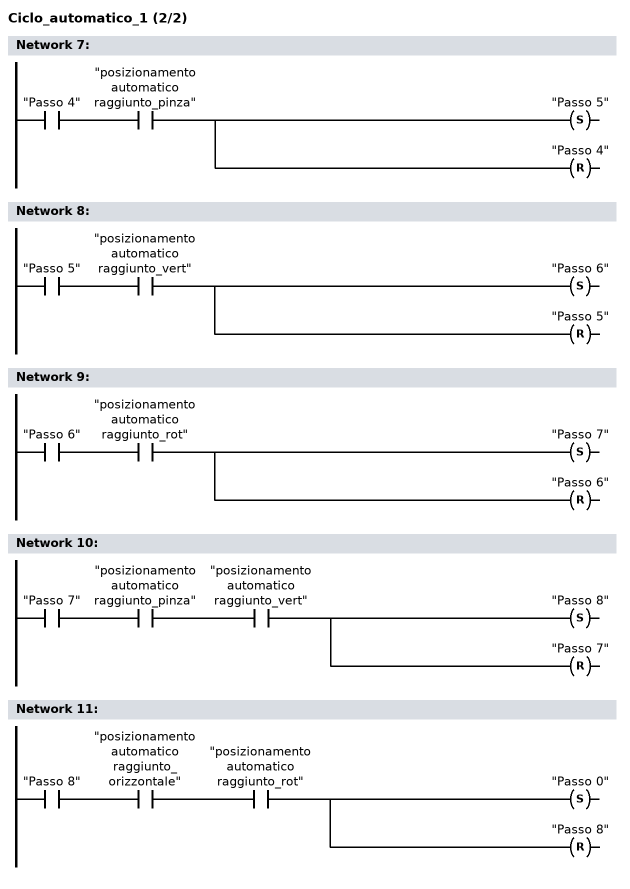
   RUNG wire#powerrail
      Contact( "Passo 4" )
      Contact( "posizionamento automatico raggiunto_pinza" )
      wire#w1
      S_Coil( "Passo 5" )
   END_RUNG
   RUNG wire#w1
      R_Coil( "Passo 4" )
   END_RUNG
   // the same network as SCL:
   IF "Passo 4" AND "posizionamento automatico raggiunto_pinza" THEN
       "Passo 5" := TRUE;
       "Passo 4" := FALSE;
   END_IF;
END_REGION

REGION Network 8
   RUNG wire#powerrail
      Contact( "Passo 5" )
      Contact( "posizionamento automatico raggiunto_vert" )
      wire#w1
      S_Coil( "Passo 6" )
   END_RUNG
   RUNG wire#w1
      R_Coil( "Passo 5" )
   END_RUNG
   // the same network as SCL:
   IF "Passo 5" AND "posizionamento automatico raggiunto_vert" THEN
       "Passo 6" := TRUE;
       "Passo 5" := FALSE;
   END_IF;
END_REGION

REGION Network 9
   RUNG wire#powerrail
      Contact( "Passo 6" )
      Contact( "posizionamento automatico raggiunto_rot" )
      wire#w1
      S_Coil( "Passo 7" )
   END_RUNG
   RUNG wire#w1
      R_Coil( "Passo 6" )
   END_RUNG
   // the same network as SCL:
   IF "Passo 6" AND "posizionamento automatico raggiunto_rot" THEN
       "Passo 7" := TRUE;
       "Passo 6" := FALSE;
   END_IF;
END_REGION

REGION Network 10
   RUNG wire#powerrail
      Contact( "Passo 7" )
      Contact( "posizionamento automatico raggiunto_pinza" )
      Contact( "posizionamento automatico raggiunto_vert" )
      wire#w1
      S_Coil( "Passo 8" )
   END_RUNG
   RUNG wire#w1
      R_Coil( "Passo 7" )
   END_RUNG
   // the same network as SCL:
   IF "Passo 7" AND "posizionamento automatico raggiunto_pinza" AND "posizionamento automatico raggiunto_vert" THEN
       "Passo 8" := TRUE;
       "Passo 7" := FALSE;
   END_IF;
END_REGION

REGION Network 11
   RUNG wire#powerrail
      Contact( "Passo 8" )
      Contact( "posizionamento automatico raggiunto_orizzontale" )
      Contact( "posizionamento automatico raggiunto_rot" )
      wire#w1
      S_Coil( "Passo 0" )
   END_RUNG
   RUNG wire#w1
      R_Coil( "Passo 8" )
   END_RUNG
   // the same network as SCL:
   IF "Passo 8" AND "posizionamento automatico raggiunto_orizzontale" AND "posizionamento automatico raggiunto_rot" THEN
       "Passo 0" := TRUE;
       "Passo 8" := FALSE;
   END_IF;
END_REGION
END_FUNCTION

FUNCTION "Ciclo_automatico_Luca_Tommy" : Void   // FC18, LAD
{ S7_Optimized_Access := 'TRUE' }
VERSION : 0.1
BEGIN

REGION Network 1
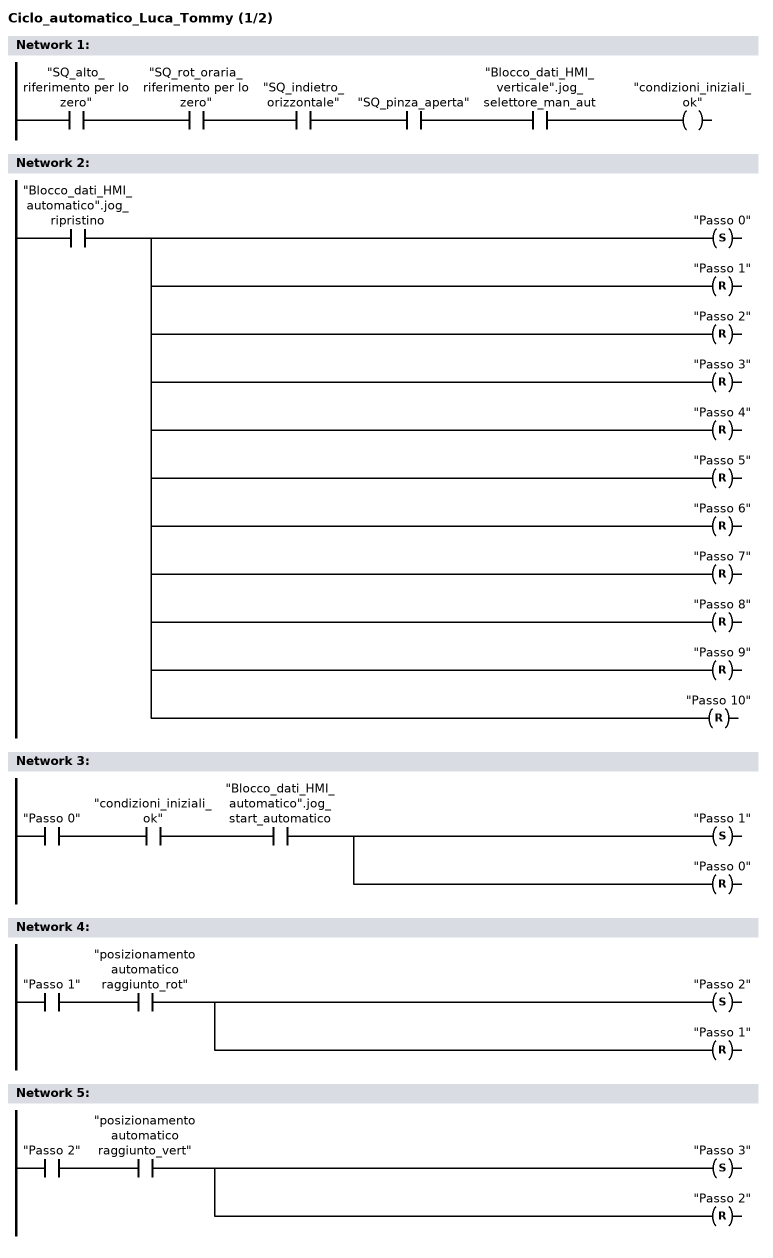
   RUNG wire#powerrail
      Contact( "SQ_alto_riferimento per lo zero" )
      Contact( "SQ_rot_oraria_riferimento per lo zero" )
      Contact( "SQ_indietro_orizzontale" )
      Contact( "SQ_pinza_aperta" )
      Contact( "Blocco_dati_HMI_verticale".jog_selettore_man_aut )
      Coil( "condizioni_iniziali_ok" )
   END_RUNG
   // the same network as SCL:
   "condizioni_iniziali_ok" := "SQ_alto_riferimento per lo zero" AND "SQ_rot_oraria_riferimento per lo zero" AND "SQ_indietro_orizzontale" AND "SQ_pinza_aperta" AND "Blocco_dati_HMI_verticale".jog_selettore_man_aut;
END_REGION

REGION Network 2
   RUNG wire#powerrail
      Contact( "Blocco_dati_HMI_automatico".jog_ripristino )
      wire#w1
      S_Coil( "Passo 0" )
   END_RUNG
   RUNG wire#w1
      R_Coil( "Passo 1" )
   END_RUNG
   RUNG wire#w1
      R_Coil( "Passo 2" )
   END_RUNG
   RUNG wire#w1
      R_Coil( "Passo 3" )
   END_RUNG
   RUNG wire#w1
      R_Coil( "Passo 4" )
   END_RUNG
   RUNG wire#w1
      R_Coil( "Passo 5" )
   END_RUNG
   RUNG wire#w1
      R_Coil( "Passo 6" )
   END_RUNG
   RUNG wire#w1
      R_Coil( "Passo 7" )
   END_RUNG
   RUNG wire#w1
      R_Coil( "Passo 8" )
   END_RUNG
   RUNG wire#w1
      R_Coil( "Passo 9" )
   END_RUNG
   RUNG wire#w1
      R_Coil( "Passo 10" )
   END_RUNG
   // the same network as SCL:
   IF "Blocco_dati_HMI_automatico".jog_ripristino THEN
       "Passo 0" := TRUE;
       "Passo 1" := FALSE;
       "Passo 2" := FALSE;
       "Passo 3" := FALSE;
       "Passo 4" := FALSE;
       "Passo 5" := FALSE;
       "Passo 6" := FALSE;
       "Passo 7" := FALSE;
       "Passo 8" := FALSE;
       "Passo 9" := FALSE;
       "Passo 10" := FALSE;
   END_IF;
END_REGION

REGION Network 3
   RUNG wire#powerrail
      Contact( "Passo 0" )
      Contact( "condizioni_iniziali_ok" )
      Contact( "Blocco_dati_HMI_automatico".jog_start_automatico )
      wire#w1
      S_Coil( "Passo 1" )
   END_RUNG
   RUNG wire#w1
      R_Coil( "Passo 0" )
   END_RUNG
   // the same network as SCL:
   IF "Passo 0" AND "condizioni_iniziali_ok" AND "Blocco_dati_HMI_automatico".jog_start_automatico THEN
       "Passo 1" := TRUE;
       "Passo 0" := FALSE;
   END_IF;
END_REGION

REGION Network 4
   RUNG wire#powerrail
      Contact( "Passo 1" )
      Contact( "posizionamento automatico raggiunto_rot" )
      wire#w1
      S_Coil( "Passo 2" )
   END_RUNG
   RUNG wire#w1
      R_Coil( "Passo 1" )
   END_RUNG
   // the same network as SCL:
   IF "Passo 1" AND "posizionamento automatico raggiunto_rot" THEN
       "Passo 2" := TRUE;
       "Passo 1" := FALSE;
   END_IF;
END_REGION

REGION Network 5
   RUNG wire#powerrail
      Contact( "Passo 2" )
      Contact( "posizionamento automatico raggiunto_vert" )
      wire#w1
      S_Coil( "Passo 3" )
   END_RUNG
   RUNG wire#w1
      R_Coil( "Passo 2" )
   END_RUNG
   // the same network as SCL:
   IF "Passo 2" AND "posizionamento automatico raggiunto_vert" THEN
       "Passo 3" := TRUE;
       "Passo 2" := FALSE;
   END_IF;
END_REGION

REGION Network 6
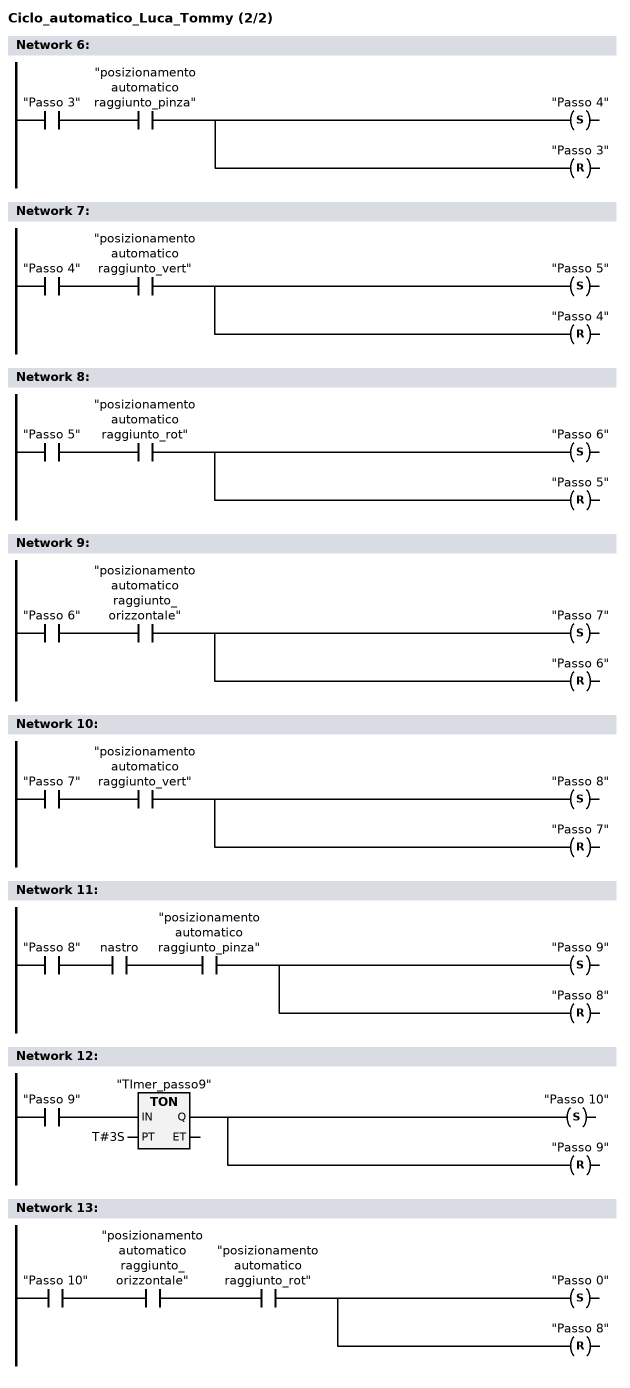
   RUNG wire#powerrail
      Contact( "Passo 3" )
      Contact( "posizionamento automatico raggiunto_pinza" )
      wire#w1
      S_Coil( "Passo 4" )
   END_RUNG
   RUNG wire#w1
      R_Coil( "Passo 3" )
   END_RUNG
   // the same network as SCL:
   IF "Passo 3" AND "posizionamento automatico raggiunto_pinza" THEN
       "Passo 4" := TRUE;
       "Passo 3" := FALSE;
   END_IF;
END_REGION

REGION Network 7
   RUNG wire#powerrail
      Contact( "Passo 4" )
      Contact( "posizionamento automatico raggiunto_vert" )
      wire#w1
      S_Coil( "Passo 5" )
   END_RUNG
   RUNG wire#w1
      R_Coil( "Passo 4" )
   END_RUNG
   // the same network as SCL:
   IF "Passo 4" AND "posizionamento automatico raggiunto_vert" THEN
       "Passo 5" := TRUE;
       "Passo 4" := FALSE;
   END_IF;
END_REGION

REGION Network 8
   RUNG wire#powerrail
      Contact( "Passo 5" )
      Contact( "posizionamento automatico raggiunto_rot" )
      wire#w1
      S_Coil( "Passo 6" )
   END_RUNG
   RUNG wire#w1
      R_Coil( "Passo 5" )
   END_RUNG
   // the same network as SCL:
   IF "Passo 5" AND "posizionamento automatico raggiunto_rot" THEN
       "Passo 6" := TRUE;
       "Passo 5" := FALSE;
   END_IF;
END_REGION

REGION Network 9
   RUNG wire#powerrail
      Contact( "Passo 6" )
      Contact( "posizionamento automatico raggiunto_orizzontale" )
      wire#w1
      S_Coil( "Passo 7" )
   END_RUNG
   RUNG wire#w1
      R_Coil( "Passo 6" )
   END_RUNG
   // the same network as SCL:
   IF "Passo 6" AND "posizionamento automatico raggiunto_orizzontale" THEN
       "Passo 7" := TRUE;
       "Passo 6" := FALSE;
   END_IF;
END_REGION

REGION Network 10
   RUNG wire#powerrail
      Contact( "Passo 7" )
      Contact( "posizionamento automatico raggiunto_vert" )
      wire#w1
      S_Coil( "Passo 8" )
   END_RUNG
   RUNG wire#w1
      R_Coil( "Passo 7" )
   END_RUNG
   // the same network as SCL:
   IF "Passo 7" AND "posizionamento automatico raggiunto_vert" THEN
       "Passo 8" := TRUE;
       "Passo 7" := FALSE;
   END_IF;
END_REGION

REGION Network 11
   RUNG wire#powerrail
      Contact( "Passo 8" )
      Contact( nastro )
      Contact( "posizionamento automatico raggiunto_pinza" )
      wire#w1
      S_Coil( "Passo 9" )
   END_RUNG
   RUNG wire#w1
      R_Coil( "Passo 8" )
   END_RUNG
   // the same network as SCL:
   IF "Passo 8" AND nastro AND "posizionamento automatico raggiunto_pinza" THEN
       "Passo 9" := TRUE;
       "Passo 8" := FALSE;
   END_IF;
END_REGION

REGION Network 12
   "TImer_passo9".TON(IN := "Passo 9", PT := T#3S);
   IF "TImer_passo9".Q THEN
       "Passo 10" := TRUE;
       "Passo 9" := FALSE;
   END_IF;
END_REGION

REGION Network 13
   RUNG wire#powerrail
      Contact( "Passo 10" )
      Contact( "posizionamento automatico raggiunto_orizzontale" )
      Contact( "posizionamento automatico raggiunto_rot" )
      wire#w1
      S_Coil( "Passo 0" )
   END_RUNG
   RUNG wire#w1
      R_Coil( "Passo 8" )
   END_RUNG
   // the same network as SCL:
   IF "Passo 10" AND "posizionamento automatico raggiunto_orizzontale" AND "posizionamento automatico raggiunto_rot" THEN
       "Passo 0" := TRUE;
       "Passo 8" := FALSE;
   END_IF;
END_REGION
END_FUNCTION

ORGANIZATION_BLOCK "Main"   // OB1, LAD, ProgramCycle
TITLE = "Main Program Sweep (Cycle)"
{ S7_Optimized_Access := 'TRUE' }
VERSION : 0.1
   VAR_INPUT
      Initial_Call : Bool;   // Initial call of this OB
      Remanence : Bool;   // =True, if remanent data are available
   END_VAR
BEGIN

REGION Network 1
